# B&R Automation Studio project CControl_Gschneitner (part 16)

#### actionUpdateStatus.st
```iecst
ACTION actionUpdateStatus:

	//Sensoren *******************************************************************************************************************************************************************************
	gStatusAnlage.FrischluftTemperatur	:= aiFrischluftTemperatur;
	gStatusAnlage.FrischluftFeuchte		:= aiFrischluftFeuchte;
	gStatusAnlage.TrockenluftTemperatur	:= aiTrockenluftTemperatur;
	gStatusAnlage.TrockenluftFeuchte	:= aiTrockenluftFeuchte;
	gStatusAnlage.AbluftFeuchte			:= aiAbluftFeuchte;
	gStatusAnlage.AbluftTemperatur		:= aiAbluftTemperatur;
	gStatusAnlage.AustrittFeuchte		:= aiAustrittFeuchte;
	gStatusAnlage.AustrittTemperatur	:= aiAustrittTemperatur;
	gStatusAnlage.DachluftFeuchte		:= aiDachluftFeuchte;
	gStatusAnlage.DachluftTemperatur	:= aiDachluftTemperatur;
	gStatusAnlage.EintrittFeuchte		:= aiEintrittFeuchte;
	gStatusAnlage.EintrittTemperatur	:= aiEintrittTemperatur;
	gStatusAnlage.HochdruckModul1		:= aiHochdruckModul1;
	gStatusAnlage.HochdruckModul2		:= aiHochdruckModul2;
	gStatusAnlage.NiederdruckModul1		:= aiNiederdruckModul1;
	gStatusAnlage.NiederdruckModul2		:= aiNiederdruckModul2;
	gStatusAnlage.Luftgeschwindigkeit	:= aiLuftgeschwindigkeit;
	gStatusAnlage.Kanaldruck			:= aiDifferenzdruck;

	//Drehzahlvorgaben *********************************************************************************************************************************************************************
	gStatusAnlage.DrehzahlKompressorModul1	:= aoDrehzahlvorgKompressorModul1;
	gStatusAnlage.DrehzahlKompressorModul2	:= aoDrehzahlvorgKompressorModul2;
	gStatusAnlage.DrehzahlVentilator1		:= aoDrehzahlvorgVentilator1;
	gStatusAnlage.DrehzahlVentilator2		:= aoDrehzahlvorgVentilator2;

	//Luftmenge Aktuell **********************************************************************************************************************************************************************
	IF Betriebsparameter.Ausstattung.Entfeuchter THEN
		gStatusAnlage.LuftmengeAktuell	:= aiLuftgeschwindigkeit * Betriebsparameter.Entfeuchter.Registerflaeche[Betriebsparameter.Entfeuchter.IndexType] * 3600;
	ELSE
		gStatusAnlage.LuftmengeAktuell	:= aiLuftgeschwindigkeit * Betriebsparameter.Allgemein.AnsaugflaecheVent * 3600;
	END_IF

	//Status Frischluftbetrieb / Umluftbetrieb *****************************************************************************************************************************************************
	IF (hmiStatus.NameSteuerung <> 4) AND (hmiStatus.NameSteuerung <> 5) THEN
		gStatusAnlage.FrischluftbetriebAktiv	:= (fbEntfUmschaltung_0.FrischluftbetriebOut AND Betriebsparameter.Umschaltklappen.Automatik) OR
		Betriebsparameter.Umschaltklappen.Frischluft;
		gStatusAnlage.UmluftbetriebAktiv		:= (fbEntfUmschaltung_0.UmluftbetriebOut AND Betriebsparameter.Umschaltklappen.Automatik) OR
		Betriebsparameter.Umschaltklappen.Umluft;
	ELSE
		gStatusAnlage.FrischluftbetriebAktiv	:= (Betriebsparameter.Umschaltklappen.Automatik AND NOT gStatusAnlage.WetterIstSchlecht) OR
		Betriebsparameter.Umschaltklappen.Frischluft;
		gStatusAnlage.UmluftbetriebAktiv		:= (Betriebsparameter.Umschaltklappen.Automatik AND gStatusAnlage.WetterIstSchlecht) OR
		Betriebsparameter.Umschaltklappen.Umluft;
	END_IF

	//Status Warmluftanforderung (Kunde Gschneitner) ***************************************************************************************************************************
	//Warmluft = Umluftklappe des jeweiligen Ventilators angesteuert (dig. Ausgang logisch 1), Kaltluft = Klappe stromlos (logisch 0).
	//Es zaehlen nur laufende Ventilatoren: steht kein laufender Ventilator auf Warmluft, wird das Heizregister wie im Stillstand behandelt.
	gStatusAnlage.Warmluft1 := hmiButtons.changeWarmluftVent1;
	gStatusAnlage.Warmluft2 := hmiButtons.changeWarmluftVent2;
	gStatusAnlage.WarmluftAnforderung := (Aktoren.VentUndKlappen.FreigabeVentilator1Out AND gStatusAnlage.Warmluft1) OR
	(Aktoren.VentUndKlappen.FreigabeVentilator2Out AND gStatusAnlage.Warmluft2);

END_ACTION
```

#### actionStillstand.st
```iecst
ACTION actionStillstand:

	gStatusAnlage.Aktor[AKTOR_SCHRITTKETTE]	:= STATUS_STILLSTAND;

	//Notstromaggregat anfordern, wenn Notbetrieb Ventilatoren noch aktiv
	Aktoren.Notstromaggregat.NotstromaggregatAngefordert := (Boxen.NotbetriebVentilator1 OR Boxen.NotbetriebVentilator2) AND
	Betriebsparameter.Ausstattung.Notstromaggregat;

	//Ölsumpfheizungen Ein, wenn Entfeuchter in Ausstattung vorhanden
	Aktoren.OelsumpfheizungModul1.Freigabe			:= Betriebsparameter.Ausstattung.Entfeuchter;
	Aktoren.OelsumpfheizungModul2.Freigabe			:= Betriebsparameter.Ausstattung.Entfeuchter AND gModul2Vorhanden;

	//Luftentfeuchter AUS
	Aktoren.KompressorModul1.Freigabe			:= FALSE;
	Aktoren.KompressorModul1.Dauerbetrieb		:= FALSE;
	Aktoren.KompressorModul1.Automatik			:= FALSE;
	Aktoren.KompressorModul1.DrehzahlvorgabeFU	:= gCmdAnlage.Leistung.DrehzahlKompressorModul1;
	Aktoren.KompressorModul2.Freigabe			:= FALSE;
	Aktoren.KompressorModul2.Dauerbetrieb		:= FALSE;
	Aktoren.KompressorModul2.Automatik			:= FALSE;
	Aktoren.KompressorModul2.DrehzahlvorgabeFU	:= gCmdAnlage.Leistung.DrehzahlKompressorModul2;

	//Entfeuchter Fremdgerät AUS
	Aktoren.EntfeuchterFremd.Freigabe		:= FALSE;
	Aktoren.EntfeuchterFremd.Dauerbetrieb	:= FALSE;
	Aktoren.EntfeuchterFremd.Automatik		:= FALSE;

	//Ventilatoren 1 freigeben bei Notbetrieb (Trocknungsgeräte noch aktiv)
	IF (Aktoren.Notstromaggregat.NotstromBereitOut OR (NOT Betriebsparameter.Ausstattung.Notstromaggregat)) THEN
		Aktoren.VentUndKlappen.AnforderungVentilator1	:= Boxen.NotbetriebVentilator1;
		Aktoren.VentUndKlappen.DrehzahlVent1Betrieb		:= gCmdAnlage.Leistung.DrehzahlVentilator1;
	END_IF

	//Ventilatoren 2 freigeben bei Notbetrieb (Trocknungsgeräte noch aktiv)
	IF (Aktoren.Notstromaggregat.NotstromBereitOut OR (NOT Betriebsparameter.Ausstattung.Notstromaggregat)) THEN
		Aktoren.VentUndKlappen.AnforderungVentilator2	:= Boxen.NotbetriebVentilator2;
		Aktoren.VentUndKlappen.DrehzahlVent2Betrieb		:= gCmdAnlage.Leistung.DrehzahlVentilator2;
	END_IF

	//Warmluftofen AUS
	Aktoren.Warmluftofen.Freigabe			:= Betriebsparameter.Ausstattung.Warmluftofen;
	Aktoren.Warmluftofen.Automatikbetrieb	:= FALSE;
	Aktoren.Warmluftofen.Dauerbetrieb		:= FALSE;

	//Heizregister AUS
	Aktoren.Heizregister.Freigabe					:= Betriebsparameter.Ausstattung.Heizregister;
	Aktoren.Heizregister.Automatikbetrieb			:= FALSE;
	Aktoren.Heizregister.Dauerbetrieb				:= FALSE;
	Aktoren.Heizregister.DrehzahlHeizregisterSoll	:= gCmdAnlage.Leistung.DrehzahlHeizregister;

	//Abluftklappe Handbetrieb
	Aktoren.Abluftklappe.Freigabe			:= Betriebsparameter.Ausstattung.Abluftklappe;
	Aktoren.Abluftklappe.Automatik			:= FALSE;
	Aktoren.Abluftklappe.Oeffnen			:= Betriebsparameter.Abluftklappe.Oeffnen;
	Aktoren.Abluftklappe.Schliessen			:= Betriebsparameter.Abluftklappe.Schliessen;

	//Abluftventilator ein, wenn Ventilator noch in Betrieb
	Aktoren.Abluftventilator.Freigabe		:= Betriebsparameter.Ausstattung.Abluftventilator AND
	(Aktoren.VentUndKlappen.Ventilator1InBetrieb OR Aktoren.VentUndKlappen.Ventilator2InBetrieb);
	Aktoren.Abluftventilator.Automatik		:= Betriebsparameter.Abluftventilator.Automatik;
	Aktoren.Abluftventilator.Ein			:= Betriebsparameter.Abluftventilator.Ein;
	Aktoren.Abluftventilator.DrehzahlSoll	:= gCmdAnlage.Leistung.DrehzahlAbluftventilator;

	//Brandschutzklappe freigeben, wenn in Ausstattung vorhanden und WLO/SHO in Betrieb
	Aktoren.Brandschutzklappe.Oeffnen		:= Betriebsparameter.Ausstattung.Brandschutzklappe AND
	(Aktoren.Warmluftofen.WarmluftofenAktiv OR Aktoren.Scheitholzofen.ScheitholzofenAktiv);
	Aktoren.Brandschutzklappe.Schliessen	:= NOT Aktoren.Brandschutzklappe.Oeffnen;

	//Bypassklappe Handbetrieb
	Aktoren.VentUndKlappen.BypassklappeOeffnen		:= Betriebsparameter.Ausstattung.Bypassklappe AND
	(Betriebsparameter.Bypassklappe.Automatik OR Betriebsparameter.Bypassklappe.Oeffnen);
	Aktoren.VentUndKlappen.BypassklappeSchliessen	:= Betriebsparameter.Ausstattung.Bypassklappe AND Betriebsparameter.Bypassklappe.Schliessen;

	//Umschaltklappen Handbetrieb
	//Kunde Gschneitner: Warmluft-/Kaltluftumschaltung bleibt auch im Stillstand in der vom Bediener gewaehlten Stellung,
	//weil der digitale Ausgang der Klappe unveraendert dem HMI-Button folgt.
	IF Betriebsparameter.Ausstattung.Umschaltklappe1 OR Betriebsparameter.Ausstattung.Umschaltklappe2 THEN
		Aktoren.VentUndKlappen.Umschaltkl1Oeffnen		:= Betriebsparameter.Ausstattung.Umschaltklappe1 AND gStatusAnlage.Warmluft1;
		Aktoren.VentUndKlappen.Umschaltkl1Schliessen	:= Betriebsparameter.Ausstattung.Umschaltklappe1 AND NOT gStatusAnlage.Warmluft1;
		Aktoren.VentUndKlappen.Umschaltkl2Oeffnen		:= Betriebsparameter.Ausstattung.Umschaltklappe2 AND gStatusAnlage.Warmluft2;
		Aktoren.VentUndKlappen.Umschaltkl2Schliessen	:= Betriebsparameter.Ausstattung.Umschaltklappe2 AND NOT gStatusAnlage.Warmluft2;
	ELSE
		Aktoren.VentUndKlappen.Umschaltkl1Schliessen		:= FALSE;
		Aktoren.VentUndKlappen.Umschaltkl2Schliessen		:= FALSE;
		Aktoren.VentUndKlappen.Umschaltkl1Oeffnen			:= FALSE;
		Aktoren.VentUndKlappen.Umschaltkl2Oeffnen			:= FALSE;
	END_IF

	//Originallogik (Stellung je nach Betriebsart / Ausstattungsmenue) - fuer Kunde Gschneitner nicht in Verwendung:
	(*
	//Umschaltklappen Handbetrieb
	IF Betriebsparameter.Ausstattung.Umschaltklappe1 OR Betriebsparameter.Ausstattung.Umschaltklappe2 THEN
		//Stellung Umluftklappen je nach Einstellung im Ausstattungsmenü
		IF Betriebsparameter.Umschaltklappen.Automatik THEN
			Aktoren.VentUndKlappen.Umschaltkl1Schliessen	:= Betriebsparameter.Ausstattung.Umschaltklappe1 AND Betriebsparameter.Ausstattung.StellungUmluftklappe1Stillstand;
			Aktoren.VentUndKlappen.Umschaltkl2Schliessen	:= Betriebsparameter.Ausstattung.Umschaltklappe2 AND Betriebsparameter.Ausstattung.StellungUmluftklappe2Stillstand;
			Aktoren.VentUndKlappen.Umschaltkl1Oeffnen		:= Betriebsparameter.Ausstattung.Umschaltklappe1 AND NOT Betriebsparameter.Ausstattung.StellungUmluftklappe1Stillstand;
			Aktoren.VentUndKlappen.Umschaltkl2Oeffnen		:= Betriebsparameter.Ausstattung.Umschaltklappe2 AND NOT Betriebsparameter.Ausstattung.StellungUmluftklappe2Stillstand;
		ELSIF Betriebsparameter.Umschaltklappen.Frischluft THEN
			Aktoren.VentUndKlappen.Umschaltkl1Schliessen	:= Betriebsparameter.Ausstattung.Umschaltklappe1;
			Aktoren.VentUndKlappen.Umschaltkl2Schliessen	:= Betriebsparameter.Ausstattung.Umschaltklappe2;
			Aktoren.VentUndKlappen.Umschaltkl1Oeffnen		:= FALSE;
			Aktoren.VentUndKlappen.Umschaltkl2Oeffnen		:= FALSE;
		ELSIF Betriebsparameter.Umschaltklappen.Umluft THEN
			Aktoren.VentUndKlappen.Umschaltkl1Schliessen	:= FALSE;
			Aktoren.VentUndKlappen.Umschaltkl2Schliessen	:= FALSE;
			Aktoren.VentUndKlappen.Umschaltkl1Oeffnen		:= Betriebsparameter.Ausstattung.Umschaltklappe1;
			Aktoren.VentUndKlappen.Umschaltkl2Oeffnen		:= Betriebsparameter.Ausstattung.Umschaltklappe2;
		END_IF
	ELSE
		Aktoren.VentUndKlappen.Umschaltkl1Schliessen		:= FALSE;
		Aktoren.VentUndKlappen.Umschaltkl2Schliessen		:= FALSE;
		Aktoren.VentUndKlappen.Umschaltkl1Oeffnen			:= FALSE;
		Aktoren.VentUndKlappen.Umschaltkl2Oeffnen			:= FALSE;
	END_IF
	*)

END_ACTION
```

#### actionBetrieb.st
```iecst
ACTION actionBetrieb:

	gStatusAnlage.Aktor[AKTOR_SCHRITTKETTE]	:= STATUS_ANLAGE_IN_BETRIEB;

	//Notstromaggregat anfordern, wenn in Box in Betrieb und in Ausstattung vorhanden
	Aktoren.Notstromaggregat.NotstromaggregatAngefordert := (Boxen.Box1Out.BoxAktiv OR Boxen.Box2Out.BoxAktiv OR Boxen.Box3Out.BoxAktiv OR
	Boxen.Box4Out.BoxAktiv OR Boxen.Box5Out.BoxAktiv OR Boxen.Box6Out.BoxAktiv OR Boxen.NotbetriebBox1 OR Boxen.NotbetriebBox2 OR
	Boxen.NotbetriebBox3 OR Boxen.NotbetriebBox4 OR Boxen.NotbetriebBox5 OR Boxen.NotbetriebBox6 OR Boxen.NotbetriebVentilator1 OR Boxen.NotbetriebVentilator2)
	AND Betriebsparameter.Ausstattung.Notstromaggregat;

	//Ölsumpfheizungen Ein, wenn Kompressoren nicht in Betrieb (und Entfeuchter in Ausstattung vorhanden)
	Aktoren.OelsumpfheizungModul1.Freigabe			:= Betriebsparameter.Ausstattung.Entfeuchter AND NOT Aktoren.KompressorModul1.FreigabeKompressorOut;
	Aktoren.OelsumpfheizungModul2.Freigabe			:= Betriebsparameter.Ausstattung.Entfeuchter AND NOT Aktoren.KompressorModul2.FreigabeKompressorOut;

	//Luftentfeuchter freigeben, wenn von Boxen angefordert und Mindestlaufzeit Ölsumpfheizung abgelaufen und Notstromaggregat bereit und Ventilator bereit
	IF (gMindestlaufzOelsumpfOk OR ((hmiStatus.CurUserLevel > 2) AND (Nutzungsdaten.BstGes.Kompressor1Std < CONST_ZEIT_TESTPHASE))) AND
		(Aktoren.Notstromaggregat.NotstromBereitOut OR (NOT Betriebsparameter.Ausstattung.Notstromaggregat)) THEN

		Aktoren.KompressorModul1.Freigabe			:= Betriebsparameter.Ausstattung.Entfeuchter AND (Boxen.FreigabeLuftentfeuchter OR Boxen.FreigabeEntfeuchterInselbetrieb) AND
		((Boxen.EntfeuchterVonVent1Abhaengig AND Boxen.FreigabeVentilator1 (*Aktoren.VentUndKlappen.FreigabeVentilator1Out*) AND NOT Aktoren.VentUndKlappen.FehlerFuVentilator1) OR
		(Boxen.EntfeuchterVonVent2Abhaengig AND Boxen.FreigabeVentilator2 (*Aktoren.VentUndKlappen.FreigabeVentilator2Out*) AND NOT Aktoren.VentUndKlappen.FehlerFuVentilator2) OR
		(Boxen.FreigabeEntfeuchterInselbetrieb AND Aktoren.VentUndKlappen.Ventilator1InBetrieb)) AND NOT
		gCmdAnlage.FehlerModul1 AND (gStatusAnlage.UmluftbetriebAktiv OR (NOT Betriebsparameter.Ausstattung.EntfeuchterNurImUmluftbetrieb)) AND NOT
		Tarifabschaltung.TarifabschaltungLuftaufbEin;
		Aktoren.KompressorModul1.Dauerbetrieb		:= Betriebsparameter.Entfeuchter.Dauerbetrieb OR Boxen.FreigabeEntfeuchterInselbetrieb;
		Aktoren.KompressorModul1.Automatik			:= Betriebsparameter.Entfeuchter.Automatikbetrieb AND NOT Boxen.FreigabeEntfeuchterInselbetrieb;
		Aktoren.KompressorModul1.DrehzahlvorgabeFU	:= gCmdAnlage.Leistung.DrehzahlKompressorModul1;

		Aktoren.KompressorModul2.Freigabe			:= (Betriebsparameter.Ausstattung.Entfeuchter AND gModul2Vorhanden) AND (Boxen.FreigabeLuftentfeuchter OR Boxen.FreigabeEntfeuchterInselbetrieb) AND
		((Boxen.EntfeuchterVonVent1Abhaengig AND Boxen.FreigabeVentilator1 (*Aktoren.VentUndKlappen.FreigabeVentilator1Out*) AND NOT Aktoren.VentUndKlappen.FehlerFuVentilator1) OR
		(Boxen.EntfeuchterVonVent2Abhaengig AND Boxen.FreigabeVentilator2 (*Aktoren.VentUndKlappen.FreigabeVentilator2Out*) AND NOT Aktoren.VentUndKlappen.FehlerFuVentilator2) OR
		(Boxen.FreigabeEntfeuchterInselbetrieb AND Aktoren.VentUndKlappen.Ventilator1InBetrieb)) AND NOT
		gCmdAnlage.FehlerModul2 AND (gStatusAnlage.UmluftbetriebAktiv OR (NOT Betriebsparameter.Ausstattung.EntfeuchterNurImUmluftbetrieb)) AND NOT
		Tarifabschaltung.TarifabschaltungLuftaufbEin;;
		Aktoren.KompressorModul2.Dauerbetrieb		:= Betriebsparameter.Entfeuchter.Dauerbetrieb OR Boxen.FreigabeEntfeuchterInselbetrieb;
		Aktoren.KompressorModul2.Automatik			:= Betriebsparameter.Entfeuchter.Automatikbetrieb AND NOT Boxen.FreigabeEntfeuchterInselbetrieb;
		Aktoren.KompressorModul2.DrehzahlvorgabeFU	:= gCmdAnlage.Leistung.DrehzahlKompressorModul2;
	END_IF

	//Entfeuchter Fremdgerät freigeben, wenn Notstromaggregat bereit (oder kein Notstromaggregat vorhanden)
	IF (Aktoren.Notstromaggregat.NotstromBereitOut OR (NOT Betriebsparameter.Ausstattung.Notstromaggregat)) THEN
		Aktoren.EntfeuchterFremd.Freigabe			:= (Boxen.FreigabeLuftentfeuchter OR Boxen.FreigabeEntfeuchterInselbetrieb) AND
		((Boxen.EntfeuchterVonVent1Abhaengig AND Boxen.FreigabeVentilator1 AND NOT Aktoren.VentUndKlappen.FehlerFuVentilator1) OR
		(Boxen.EntfeuchterVonVent2Abhaengig AND Boxen.FreigabeVentilator2 AND NOT Aktoren.VentUndKlappen.FehlerFuVentilator2) OR
		(Boxen.FreigabeEntfeuchterInselbetrieb AND Aktoren.VentUndKlappen.Ventilator1InBetrieb)) AND NOT
		gCmdAnlage.FehlerModul1 AND (gStatusAnlage.UmluftbetriebAktiv OR (NOT Betriebsparameter.Ausstattung.EntfeuchterNurImUmluftbetrieb)) AND NOT
		Tarifabschaltung.TarifabschaltungLuftaufbEin;
		Aktoren.EntfeuchterFremd.Dauerbetrieb		:= Betriebsparameter.Entfeuchter.Dauerbetrieb OR Boxen.FreigabeEntfeuchterInselbetrieb;
		Aktoren.EntfeuchterFremd.Automatik			:= Betriebsparameter.Entfeuchter.Automatikbetrieb AND NOT Boxen.FreigabeEntfeuchterInselbetrieb;
	ELSE
		Aktoren.EntfeuchterFremd.Freigabe		:= FALSE;
		Aktoren.EntfeuchterFremd.Dauerbetrieb	:= FALSE;
		Aktoren.EntfeuchterFremd.Automatik		:= FALSE;
	END_IF

	//Ventilatoren 1 freigeben, wenn von Boxen angefordert und keine Tarifabschaltung (ausgenommen bei Notbetrieb wenn Trocknungsgeräte noch aktiv)
	IF (Aktoren.Notstromaggregat.NotstromBereitOut OR (NOT Betriebsparameter.Ausstattung.Notstromaggregat)) THEN
		Aktoren.VentUndKlappen.AnforderungVentilator1	:= (Boxen.FreigabeVentilator1 OR Boxen.NotbetriebVentilator1) AND NOT
		(Tarifabschaltung.TarifabschaltungEin AND NOT Boxen.NotbetriebVentilator1);
		Aktoren.VentUndKlappen.DrehzahlVent1Betrieb		:= gCmdAnlage.Leistung.DrehzahlVentilator1;
	ELSE
		Aktoren.VentUndKlappen.AnforderungVentilator1	:= FALSE;
	END_IF

	//Ventilatoren 2 freigeben, wenn von Boxen angefordert und keine Tarifabschaltung (ausgenommen bei Notbetrieb wenn Trocknungsgeräte noch aktiv)
	IF (Aktoren.Notstromaggregat.NotstromBereitOut OR (NOT Betriebsparameter.Ausstattung.Notstromaggregat)) THEN
		Aktoren.VentUndKlappen.AnforderungVentilator2	:= (Boxen.FreigabeVentilator2 OR Boxen.NotbetriebVentilator2) AND NOT
		(Tarifabschaltung.TarifabschaltungEin AND NOT Boxen.NotbetriebVentilator2);
		Aktoren.VentUndKlappen.DrehzahlVent2Betrieb		:= gCmdAnlage.Leistung.DrehzahlVentilator2;
	ELSE
		Aktoren.VentUndKlappen.AnforderungVentilator2	:= FALSE;
	END_IF

	//Warmluftofen freigeben, wenn von Boxen angefordert und Ventilator in Betrieb
	Aktoren.Warmluftofen.Freigabe			:= Betriebsparameter.Ausstattung.Warmluftofen AND Boxen.FreigabeWarmluftofen AND
	((Boxen.WarmluftofenVonVent1Abhaengig AND Aktoren.VentUndKlappen.FreigabeVentilator1Out AND NOT Aktoren.VentUndKlappen.FehlerFuVentilator1) OR
	(Boxen.WarmluftofenVonVent2Abhaengig AND Aktoren.VentUndKlappen.FreigabeVentilator2Out AND NOT Aktoren.VentUndKlappen.FehlerFuVentilator2)) AND NOT
	Tarifabschaltung.TarifabschaltungLuftaufbEin;
	Aktoren.Warmluftofen.Automatikbetrieb	:= Betriebsparameter.Warmluftofen.AutomatikbetriebEin;
	Aktoren.Warmluftofen.Dauerbetrieb		:= Betriebsparameter.Warmluftofen.DauerbetriebEin;

	//Heizregister freigeben, wenn von Boxen angefordert und zuständiger Ventilator aktiv
	Aktoren.Heizregister.Freigabe					:= Betriebsparameter.Ausstattung.Heizregister AND Boxen.FreigabeHeizregister  AND
	((Boxen.HeizregisterVonVent1Abhaengig AND Aktoren.VentUndKlappen.FreigabeVentilator1Out AND NOT Aktoren.VentUndKlappen.FehlerFuVentilator1) OR
	(Boxen.HeizregisterVonVent2Abhaengig AND Aktoren.VentUndKlappen.FreigabeVentilator2Out AND NOT Aktoren.VentUndKlappen.FehlerFuVentilator2)) AND NOT
	Tarifabschaltung.TarifabschaltungLuftaufbEin;
	Aktoren.Heizregister.Automatikbetrieb			:= Betriebsparameter.Heizregister.AutomatikbetriebEin;
	Aktoren.Heizregister.Dauerbetrieb				:= Betriebsparameter.Heizregister.DauerbetriebEin;
	Aktoren.Heizregister.DrehzahlHeizregisterSoll	:= gCmdAnlage.Leistung.DrehzahlHeizregister;

	//Kunde Gschneitner: Heizregister abschalten, wenn kein laufender Ventilator auf Warmluft steht.
	//Der Baustein wird dabei exakt wie im Stillstand versorgt -> FreigabeHeizregisterOut = FALSE und DrehzahlHeizregisterOut = 0.0.
	IF NOT gStatusAnlage.WarmluftAnforderung THEN
		Aktoren.Heizregister.Automatikbetrieb			:= FALSE;
		Aktoren.Heizregister.Dauerbetrieb				:= FALSE;
		Aktoren.Heizregister.DrehzahlHeizregisterSoll	:= 0.0;
	END_IF

	//Abluftklappe freigeben, wenn in Ausstattung vorhanden
	Aktoren.Abluftklappe.Freigabe			:= Betriebsparameter.Ausstattung.Abluftklappe;
	Aktoren.Abluftklappe.Automatik			:= Betriebsparameter.Abluftklappe.Automatik AND NOT
	(gStatusAnlage.FrischluftbetriebAktiv AND Betriebsparameter.Ausstattung.AbluftklImFrischlbetrImmerOffen);
	Aktoren.Abluftklappe.Oeffnen			:= Betriebsparameter.Abluftklappe.Oeffnen OR
	(gStatusAnlage.FrischluftbetriebAktiv AND Betriebsparameter.Ausstattung.AbluftklImFrischlbetrImmerOffen AND NOT Betriebsparameter.Abluftklappe.Schliessen);
	Aktoren.Abluftklappe.Schliessen			:= Betriebsparameter.Abluftklappe.Schliessen;

	//Abluftventilator freigeben, wenn in Ausstattung vorhanden
	Aktoren.Abluftventilator.Freigabe		:= Betriebsparameter.Ausstattung.Abluftventilator;
	Aktoren.Abluftventilator.Automatik		:= Betriebsparameter.Abluftventilator.Automatik AND (Boxen.Box1Out.BoxAktiv OR Boxen.Box2Out.BoxAktiv OR
	Boxen.Box3Out.BoxAktiv OR Boxen.Box4Out.BoxAktiv OR Boxen.Box5Out.BoxAktiv OR Boxen.Box6Out.BoxAktiv) AND NOT
	(gStatusAnlage.FrischluftbetriebAktiv AND Betriebsparameter.Ausstattung.AbluftklImFrischlbetrImmerOffen);
	Aktoren.Abluftventilator.Ein			:= Betriebsparameter.Abluftventilator.Ein OR
	(gStatusAnlage.FrischluftbetriebAktiv AND Betriebsparameter.Ausstattung.AbluftklImFrischlbetrImmerOffen AND (Boxen.Box1Out.BoxAktiv OR Boxen.Box2Out.BoxAktiv OR
	Boxen.Box3Out.BoxAktiv OR Boxen.Box4Out.BoxAktiv OR Boxen.Box5Out.BoxAktiv OR Boxen.Box6Out.BoxAktiv));
	Aktoren.Abluftventilator.DrehzahlSoll	:= gCmdAnlage.Leistung.DrehzahlAbluftventilator;

	//Brandschutzklappe freigeben, wenn in Ausstattung vorhanden und WLO/SHO in Betrieb
	Aktoren.Brandschutzklappe.Oeffnen		:= Betriebsparameter.Ausstattung.Brandschutzklappe AND
	(Aktoren.Warmluftofen.WarmluftofenAktiv OR Aktoren.Scheitholzofen.ScheitholzofenAktiv);
	Aktoren.Brandschutzklappe.Schliessen	:= NOT Aktoren.Brandschutzklappe.Oeffnen;

	//Bypassklappe freigeben, wenn in Ausstattung vorhanden
	IF Betriebsparameter.Bypassklappe.Automatik AND Betriebsparameter.Ausstattung.Bypassklappe AND NOT Betriebsparameter.Ausstattung.EntfeuchterFremd THEN
		IF NOT Aktoren.KompressorModul1.Freigabe AND NOT Aktoren.KompressorModul2.Freigabe THEN
			Aktoren.VentUndKlappen.BypassklappeOeffnen		:= TRUE;
			Aktoren.VentUndKlappen.BypassklappeSchliessen	:= FALSE;
		ELSE
			Aktoren.VentUndKlappen.BypassklappeOeffnen		:=  NOT Aktoren.KompressorModul1.loc_StatusFeuchteOk AND NOT Aktoren.KompressorModul2.loc_StatusFeuchteOk;
			Aktoren.VentUndKlappen.BypassklappeSchliessen	:= Aktoren.KompressorModul1.loc_StatusFeuchteOk OR Aktoren.KompressorModul2.loc_StatusFeuchteOk;
		END_IF
	//Ausstattung mit Entfeuchter Fremdgerät
	ELSIF Betriebsparameter.Bypassklappe.Automatik AND Betriebsparameter.Ausstattung.Bypassklappe THEN
		IF NOT Aktoren.EntfeuchterFremd.Freigabe THEN
			Aktoren.VentUndKlappen.BypassklappeOeffnen		:= TRUE;
			Aktoren.VentUndKlappen.BypassklappeSchliessen	:= FALSE;
		ELSE
			Aktoren.VentUndKlappen.BypassklappeOeffnen		:=  NOT Aktoren.EntfeuchterFremd.WitterungIstSchlecht;
			Aktoren.VentUndKlappen.BypassklappeSchliessen	:= Aktoren.EntfeuchterFremd.WitterungIstSchlecht;
		END_IF
	ELSE
		Aktoren.VentUndKlappen.BypassklappeOeffnen		:= Betriebsparameter.Ausstattung.Bypassklappe AND Betriebsparameter.Bypassklappe.Oeffnen;
		Aktoren.VentUndKlappen.BypassklappeSchliessen	:= Betriebsparameter.Ausstattung.Bypassklappe AND Betriebsparameter.Bypassklappe.Schliessen;
	END_IF
	(*
	Aktoren.VentUndKlappen.BypassklappeOeffnen		:= Betriebsparameter.Ausstattung.Bypassklappe AND (Betriebsparameter.Bypassklappe.Oeffnen OR
	(Betriebsparameter.Bypassklappe.Automatik AND NOT Aktoren.KompressorModul1.loc_StatusFeuchteOk AND NOT Aktoren.KompressorModul2.loc_StatusFeuchteOk));
	Aktoren.VentUndKlappen.BypassklappeSchliessen	:= Betriebsparameter.Ausstattung.Bypassklappe AND (Betriebsparameter.Bypassklappe.Schliessen OR
	(Betriebsparameter.Bypassklappe.Automatik AND (Aktoren.KompressorModul1.loc_StatusFeuchteOk OR Aktoren.KompressorModul2.loc_StatusFeuchteOk)));
	*)

	//Umschaltklappen je nach Betriebsart umschalten
	//Kunde Gschneitner: die Umschaltklappen werden als Warmluft-/Kaltluftumschaltung verwendet und direkt vom Bediener geschaltet.
	//Die Betriebsart ist fest auf Frischluft gestellt, deshalb entfaellt die witterungsgefuehrte Umschaltung.
	//Die Klappenbausteine werden hier mit der tatsaechlichen Stellung versorgt, damit Laufzeit-/Endlagenueberwachung und
	//die Statusanzeigen in der Visu mit dem realen Ausgang zusammenpassen.
	IF Betriebsparameter.Ausstattung.Umschaltklappe1 OR Betriebsparameter.Ausstattung.Umschaltklappe2 THEN
		Aktoren.VentUndKlappen.Umschaltkl1Oeffnen		:= Betriebsparameter.Ausstattung.Umschaltklappe1 AND gStatusAnlage.Warmluft1;
		Aktoren.VentUndKlappen.Umschaltkl1Schliessen	:= Betriebsparameter.Ausstattung.Umschaltklappe1 AND NOT gStatusAnlage.Warmluft1;
		Aktoren.VentUndKlappen.Umschaltkl2Oeffnen		:= Betriebsparameter.Ausstattung.Umschaltklappe2 AND gStatusAnlage.Warmluft2;
		Aktoren.VentUndKlappen.Umschaltkl2Schliessen	:= Betriebsparameter.Ausstattung.Umschaltklappe2 AND NOT gStatusAnlage.Warmluft2;
	ELSE
		Aktoren.VentUndKlappen.Umschaltkl1Schliessen		:= FALSE;
		Aktoren.VentUndKlappen.Umschaltkl2Schliessen		:= FALSE;
		Aktoren.VentUndKlappen.Umschaltkl1Oeffnen			:= FALSE;
		Aktoren.VentUndKlappen.Umschaltkl2Oeffnen			:= FALSE;
	END_IF

	//Originallogik (Betriebsart Automatik/Frischluft/Umluft) - fuer Kunde Gschneitner nicht in Verwendung:
	(*
	//Umschaltklappen je nach Betriebsart umschalten
	IF Betriebsparameter.Ausstattung.Umschaltklappe1 OR Betriebsparameter.Ausstattung.Umschaltklappe2 THEN
		//Konfiguration HB3000 und HB4000 -> Umschaltklappen nach Witterung umschalten (Kein eigener Schaltpunkt)
		IF (hmiStatus.NameSteuerung = 4) OR (hmiStatus.NameSteuerung = 5) THEN
			IF Betriebsparameter.Umschaltklappen.Frischluft OR (Betriebsparameter.Umschaltklappen.Automatik AND NOT gStatusAnlage.WetterIstSchlecht) THEN
				Aktoren.VentUndKlappen.Umschaltkl1Schliessen	:= Betriebsparameter.Ausstattung.Umschaltklappe1;
				Aktoren.VentUndKlappen.Umschaltkl2Schliessen	:= Betriebsparameter.Ausstattung.Umschaltklappe2;
				Aktoren.VentUndKlappen.Umschaltkl1Oeffnen		:= FALSE;
				Aktoren.VentUndKlappen.Umschaltkl2Oeffnen		:= FALSE;
			ELSIF Betriebsparameter.Umschaltklappen.Umluft OR (Betriebsparameter.Umschaltklappen.Automatik AND gStatusAnlage.WetterIstSchlecht) THEN
				Aktoren.VentUndKlappen.Umschaltkl1Schliessen	:= FALSE;
				Aktoren.VentUndKlappen.Umschaltkl2Schliessen	:= FALSE;
				Aktoren.VentUndKlappen.Umschaltkl1Oeffnen		:= Betriebsparameter.Ausstattung.Umschaltklappe1;
				Aktoren.VentUndKlappen.Umschaltkl2Oeffnen		:= Betriebsparameter.Ausstattung.Umschaltklappe2;
			END_IF
		ELSIF Betriebsparameter.Umschaltklappen.Frischluft OR (Betriebsparameter.Umschaltklappen.Automatik AND gStatusAnlage.FrischluftbetriebAktiv) THEN
			Aktoren.VentUndKlappen.Umschaltkl1Schliessen	:= Betriebsparameter.Ausstattung.Umschaltklappe1;
			Aktoren.VentUndKlappen.Umschaltkl2Schliessen	:= Betriebsparameter.Ausstattung.Umschaltklappe2;
			Aktoren.VentUndKlappen.Umschaltkl1Oeffnen		:= FALSE;
			Aktoren.VentUndKlappen.Umschaltkl2Oeffnen		:= FALSE;
		ELSIF Betriebsparameter.Umschaltklappen.Umluft OR (Betriebsparameter.Umschaltklappen.Automatik AND gStatusAnlage.UmluftbetriebAktiv) THEN
			Aktoren.VentUndKlappen.Umschaltkl1Schliessen	:= FALSE;
			Aktoren.VentUndKlappen.Umschaltkl2Schliessen	:= FALSE;
			Aktoren.VentUndKlappen.Umschaltkl1Oeffnen		:= Betriebsparameter.Ausstattung.Umschaltklappe1;
			Aktoren.VentUndKlappen.Umschaltkl2Oeffnen		:= Betriebsparameter.Ausstattung.Umschaltklappe2;
		END_IF
	ELSE
		Aktoren.VentUndKlappen.Umschaltkl1Schliessen		:= FALSE;
		Aktoren.VentUndKlappen.Umschaltkl2Schliessen		:= FALSE;
		Aktoren.VentUndKlappen.Umschaltkl1Oeffnen			:= FALSE;
		Aktoren.VentUndKlappen.Umschaltkl2Oeffnen			:= FALSE;
	END_IF
	*)

END_ACTION
```

### Package Logical/Steuerung - Generierung der Start- und Stoppsignale

### Program Logical/Steuerung/StartStopp (IEC) - Auswertung der Start- und Stoppsignale

#### StartStopp.st - Zyklischer Code
```iecst
PROGRAM _CYCLIC

	//Ticks erzeugen
	//==============
	fbLascoZdxx_0(IN	:= Echtzeit.Milli / 100);
	hmilliTick			:= fbLascoZdxx_0.Q;

	fbLascoPuge_0(StartMitPuls := TRUE, Tick := hmilliTick, ZeitPuls := 8, ZeitPause := 8,);
	hmiBlink			:= fbLascoPuge_0.PulsQ;

	//Automatik oder Testmodus
	//************************

	gCmdAnlage.Auto   		:= NOT hmiButtons.TestbetriebEin;
	gCmdAnlage.Test   		:= hmiButtons.TestbetriebEin;

	//Externe Start/Stopp- Signale
(*	gCmdAnlage.StartExtern		:= diAnfEntfeuchterExtern;
	gCmdAnlage.StoppExtern		:= NOT diAnfEntfeuchterExtern;*)

	//Start- und Stoppsignale auswerten
	//=================================

	//Startsignal geben, wenn eine der Boxen angefordert wird
	gCmdAnlage.Start	:= gCmdAnlage.Auto AND (Boxen.Box1Out.BoxBereit OR Boxen.Box2Out.BoxBereit OR Boxen.Box3Out.BoxBereit OR Boxen.Box4Out.BoxBereit OR
	Boxen.Box5Out.BoxBereit OR Boxen.Box6Out.BoxBereit OR Boxen.EntfeuchterInselbetrAktivOut);

	//Stopsignal geben, wenn keine Box angefordert ist
	gCmdAnlage.Stop		:= gCmdAnlage.Auto AND NOT Boxen.Box1Out.BoxBereit AND NOT Boxen.Box2Out.BoxBereit AND NOT Boxen.Box3Out.BoxBereit AND NOT Boxen.Box4Out.BoxBereit AND NOT
	Boxen.Box5Out.BoxBereit AND NOT Boxen.Box6Out.BoxBereit AND NOT Boxen.EntfeuchterInselbetrAktivOut;

	//Signal Fehler-Stopp erzeugen (kein Start möglich bzw. Abbruch Trocknung)
	//Fehlerstopp entfernt (Trocknung lässt sich dennoch starten, je nach Fehler werden die einzelnen Aktoren nicht freigegeben
	gCmdAnlage.FehlerStopp	:= FALSE;
(*	gCmdAnlage.FehlerStopp	:= (gCmdAnlage.Auto AND (alarmFehler[FEHLER_24VDC] OR alarmFehler[FEHLER_ENDLAGEN_BOXENKLAPPE_1] OR
	alarmFehler[FEHLER_ENDLAGEN_BOXENKLAPPE_2] OR alarmFehler[FEHLER_ENDLAGEN_BOXENKLAPPE_3] OR alarmFehler[FEHLER_ENDLAGEN_BOXENKLAPPE_4] OR
	alarmFehler[FEHLER_ENDLAGEN_BOXENKLAPPE_5] OR alarmFehler[FEHLER_ENDLAGEN_BOXENKLAPPE_6] OR alarmFehler[FEHLER_ENDLAGEN_BYPASSKLAPPE] OR
	alarmFehler[FEHLER_ENDLAGEN_UMSCHALTKLAPPE1] OR alarmFehler[FEHLER_ENDLAGEN_UMSCHALTKLAPPE2] OR alarmFehler[FEHLER_IO_TEST_NICHT_FERTIG] OR
	alarmFehler[FEHLER_KOMMUNIKATION_DISPLAY_IO] OR alarmFehler[FEHLER_BETRIEBSMLDG_NOTSTROM] OR alarmFehler[FEHLER_BETRIEBSMLDG_VENTILATOR1] OR
	alarmFehler[FEHLER_BETRIEBSMLDG_VENTILATOR2]));

	//Bei Doppelmodulen Anlage nur stoppen, wenn bei beiden Modulen ein Fehler anliegt
	IF gModul2Vorhanden THEN
		gCmdAnlage.FehlerStopp := (gCmdAnlage.Auto AND (alarmFehler[FEHLER_24VDC] OR alarmFehler[FEHLER_ENDLAGEN_BOXENKLAPPE_1] OR alarmFehler[FEHLER_ENDLAGEN_BOXENKLAPPE_2] OR
		alarmFehler[FEHLER_ENDLAGEN_BOXENKLAPPE_3] OR alarmFehler[FEHLER_ENDLAGEN_BOXENKLAPPE_4] OR alarmFehler[FEHLER_ENDLAGEN_BOXENKLAPPE_5] OR
		alarmFehler[FEHLER_ENDLAGEN_BOXENKLAPPE_6] OR alarmFehler[FEHLER_ENDLAGEN_BYPASSKLAPPE] OR alarmFehler[FEHLER_ENDLAGEN_UMSCHALTKLAPPE1] OR
		alarmFehler[FEHLER_ENDLAGEN_UMSCHALTKLAPPE2] OR alarmFehler[FEHLER_IO_TEST_NICHT_FERTIG] OR alarmFehler[FEHLER_KOMMUNIKATION_DISPLAY_IO] OR
		alarmFehler[FEHLER_EINTRITT_TEMP_ZU_HOCH] OR alarmFehler[FEHLER_EINTRITT_TEMP_ZU_NIEDRIG] OR (gCmdAnlage.FehlerModul1 AND gCmdAnlage.FehlerModul2)));
	ELSE
		gCmdAnlage.FehlerStopp := (gCmdAnlage.Auto AND (alarmFehler[FEHLER_24VDC] OR alarmFehler[FEHLER_ENDLAGEN_BOXENKLAPPE_1] OR alarmFehler[FEHLER_ENDLAGEN_BOXENKLAPPE_2] OR
		alarmFehler[FEHLER_ENDLAGEN_BOXENKLAPPE_3] OR alarmFehler[FEHLER_ENDLAGEN_BOXENKLAPPE_4] OR alarmFehler[FEHLER_ENDLAGEN_BOXENKLAPPE_5] OR
		alarmFehler[FEHLER_ENDLAGEN_BOXENKLAPPE_6] OR alarmFehler[FEHLER_ENDLAGEN_BYPASSKLAPPE] OR alarmFehler[FEHLER_ENDLAGEN_UMSCHALTKLAPPE1] OR
		alarmFehler[FEHLER_ENDLAGEN_UMSCHALTKLAPPE2] OR alarmFehler[FEHLER_IO_TEST_NICHT_FERTIG] OR alarmFehler[FEHLER_KOMMUNIKATION_DISPLAY_IO] OR
		alarmFehler[FEHLER_EINTRITT_TEMP_ZU_HOCH] OR alarmFehler[FEHLER_EINTRITT_TEMP_ZU_NIEDRIG] OR gCmdAnlage.FehlerModul1));
	END_IF
	*)
	//Fehler Modul 1
	gCmdAnlage.FehlerModul1	:= (gCmdAnlage.Auto AND (alarmFehler[FEHLER_BETRIEBSMLDG_KOMPR_MOD1] OR alarmFehler[FEHLER_FU_KOMPRESSOR_MODUL1] OR alarmFehler[FEHLER_HOCHDRUCK_MODUL1] OR
	alarmFehler[FEHLER_KOPFTEMP_KOMPR_MOD1] OR alarmFehler[FEHLER_NIEDERDRUCK_MODUL1] OR alarmFehler[FEHLER_OELDRUCK_KOMPR_MOD1] OR alarmFehler[FEHLER_SENSOR_HOCHDRUCK_MOD1] OR
	alarmFehler[FEHLER_SENSOR_NIEDERDRUCK_MOD1] OR alarmFehler[FEHLER_VOLLSCHUTZ_KOMPR_MOD1] OR alarmFehler[FEHLER_LZ_PUMPDOWN_MOD1] OR alarmFehler[FEHLER_DREHFELD] OR
	alarmFehler[FEHLER_ENTF_FREMD_BETRMLDG] OR alarmFehler[FEHLER_ENTF_FREMD_STOERMELDUNG])); //Ab V2.0.0: Fehler Entfeuchter Fremd hinzugefügt

	//Fehler Modul 2
	gCmdAnlage.FehlerModul2	:= (gCmdAnlage.Auto AND gModul2Vorhanden AND (alarmFehler[FEHLER_BETRIEBSMLDG_KOMPR_MOD2] OR alarmFehler[FEHLER_FU_KOMPRESSOR_MODUL2] OR alarmFehler[FEHLER_HOCHDRUCK_MODUL2] OR
	alarmFehler[FEHLER_KOPFTEMP_KOMPR_MOD2] OR alarmFehler[FEHLER_NIEDERDRUCK_MODUL2] OR alarmFehler[FEHLER_OELDRUCK_KOMPR_MOD2] OR alarmFehler[FEHLER_SENSOR_HOCHDRUCK_MOD2] OR
	alarmFehler[FEHLER_SENSOR_NIEDERDRUCK_MOD2] OR alarmFehler[FEHLER_VOLLSCHUTZ_KOMPR_MOD2] OR alarmFehler[FEHLER_LZ_PUMPDOWN_MOD2] OR alarmFehler[FEHLER_DREHFELD]));

	//Betriebsmeldung und Störmeldung
	gStatusAnlage.Betrieb	:= gAktModus = BETRIEB;

	IF gStatusAnlage.Betrieb AND (doVentilator1Ein OR doVentilator2Ein) THEN
		doTrocknungInBetrieb := TRUE;
	ELSIF gStatusAnlage.Betrieb AND (doKompressorEinModul1 OR doKompressorEinModul2) AND NOT Betriebsparameter.Ausstattung.Ventilator1 THEN
		doTrocknungInBetrieb := TRUE;
	ELSIF gStatusAnlage.Betrieb THEN
		doTrocknungInBetrieb := hmiBlink;
	ELSE
		doTrocknungInBetrieb := FALSE;
	END_IF

	doTrocknungStoerung		:= gStatusAnlage.Fehler.SummeFehler;

END_PROGRAM
```

#### StartStopp.var - Lokale Variablen
```iecst
VAR
	fbLascoZdxx_0 : {REDUND_UNREPLICABLE} fbLascoZdxx;
	hmilliTick : {REDUND_UNREPLICABLE} BOOL;
	fbLascoPuge_0 : {REDUND_UNREPLICABLE} fbLascoPuge;
	hmiBlink : {REDUND_UNREPLICABLE} BOOL;
END_VAR
```

### Package Logical/Regelung - Luftmengen- und Druckregler

### Program Logical/Regelung/Leistung (IEC) - Leistungsvorgabe an Ventilatoren

#### Leistung.st - Zyklischer Code
```iecst
PROGRAM _INIT

	//Luftmengenregler für Ventilator 1 initialisieren
	fbPidLuftmengeVent1.Mode	:= FBREG_MODUS_AUS;
	fbPidLuftmengeVent1();

	//Luftmengenregler für Ventilator 2 initialisieren
	fbPidLuftmengeVent2.Mode	:= FBREG_MODUS_AUS;
	fbPidLuftmengeVent2();

	//Regler Entfeuchter Kompressor 1 -Drehzahl initialisieren
	fbPidKompressor1.Mode	:= FBREG_MODUS_AUS;
	fbPidKompressor1();

	//Regler Entfeuchter Kompressor 2 -Drehzahl initialisieren
	fbPidKompressor2.Mode	:= FBREG_MODUS_AUS;
	fbPidKompressor2();

	//Regler Heizregister-Pumpe initialisieren
	fbPidHeizregister.Mode	:= FBREG_MODUS_AUS;
	fbPidHeizregister();

	//Abluftregler initialisieren
	fbPidAbluftregler.Mode		:= FBREG_MODUS_AUS;
	fbPidAbluftregler();

END_PROGRAM

PROGRAM _CYCLIC

	//Zeitticks erzeugen
	fbLascoZdxx_0(IN 	:= Echtzeit.Minute);
	minTick				:= fbLascoZdxx_0.Q;
	fbLascoZdxx_1(IN	:= Echtzeit.Sekunde);
	sekTick				:= fbLascoZdxx_1.Q;

	//Erforderliche Soll-Luftmengen für Ventilator 1 & 2 ermitteln
	//************************************************************

	fbBoxenLuftmengen_0.EntfeuchterInBetrieb			:= Aktoren.KompressorModul1.FreigabeKompressorOut OR Aktoren.KompressorModul2.FreigabeKompressorOut OR
	diEntfeuchterFremdInBetrieb;
	//Kunde Gschneitner: wird weiter unten je Parametersatz (Kalt-/Warmluft) ueberschrieben
	fbBoxenLuftmengen_0.FrischluftbetriebAktiv			:= gStatusAnlage.FrischluftbetriebAktiv;
	fbBoxenLuftmengen_0.UmluftbetriebAktiv				:= gStatusAnlage.UmluftbetriebAktiv;
	fbBoxenLuftmengen_0.LuftgeschwEntfeuchterMin		:= Betriebsparameter.Entfeuchter.LuftgeschwEntfeuchterMin;
	fbBoxenLuftmengen_0.LuftgeschwEntfeuchterMax		:= Betriebsparameter.Entfeuchter.LuftgeschwEntfeuchterMax;
	fbBoxenLuftmengen_0.LuftmengeSollProM2FrischlVent1	:= Betriebsparameter.Ventilator1.LuftmengeSollFrischluft;
	fbBoxenLuftmengen_0.LuftmengeSollProM2UmluftVent1	:= Betriebsparameter.Ventilator1.LuftmengeSollUmluft;
	fbBoxenLuftmengen_0.LuftmengeSollProM2FrischlVent2	:= Betriebsparameter.Ventilator2.LuftmengeSollFrischluft;
	fbBoxenLuftmengen_0.LuftmengeSollProM2UmluftVent2	:= Betriebsparameter.Ventilator2.LuftmengeSollUmluft;
	IF Betriebsparameter.Ausstattung.EntfeuchterFremd THEN
		fbBoxenLuftmengen_0.RegisterflaecheEntfeuchter		:= Betriebsparameter.Allgemein.AnsaugflaecheVent;
	ELSE
		fbBoxenLuftmengen_0.RegisterflaecheEntfeuchter		:= Betriebsparameter.Entfeuchter.Registerflaeche[Betriebsparameter.Entfeuchter.IndexType];
	END_IF

	fbBoxenLuftmengen_0.Box1.BoxIstAktiv		:= Boxen.Box1Out.BoxAktiv;
	fbBoxenLuftmengen_0.Box1.GrundflaecheBox	:= Betriebsparameter.Boxen[1].Grundflaeche;
	fbBoxenLuftmengen_0.Box1.Ventilator1		:= Betriebsparameter.Boxen[1].Ventilator1;
	fbBoxenLuftmengen_0.Box1.Ventilator2		:= Betriebsparameter.Boxen[1].Ventilator2;

	fbBoxenLuftmengen_0.Box2.BoxIstAktiv		:= Boxen.Box2Out.BoxAktiv;
	fbBoxenLuftmengen_0.Box2.GrundflaecheBox	:= Betriebsparameter.Boxen[2].Grundflaeche;
	fbBoxenLuftmengen_0.Box2.Ventilator1		:= Betriebsparameter.Boxen[2].Ventilator1;
	fbBoxenLuftmengen_0.Box2.Ventilator2		:= Betriebsparameter.Boxen[2].Ventilator2;

	fbBoxenLuftmengen_0.Box3.BoxIstAktiv		:= Boxen.Box3Out.BoxAktiv;
	fbBoxenLuftmengen_0.Box3.GrundflaecheBox	:= Betriebsparameter.Boxen[3].Grundflaeche;
	fbBoxenLuftmengen_0.Box3.Ventilator1		:= Betriebsparameter.Boxen[3].Ventilator1;
	fbBoxenLuftmengen_0.Box3.Ventilator2		:= Betriebsparameter.Boxen[3].Ventilator2;

	fbBoxenLuftmengen_0.Box4.BoxIstAktiv		:= Boxen.Box4Out.BoxAktiv;
	fbBoxenLuftmengen_0.Box4.GrundflaecheBox	:= Betriebsparameter.Boxen[4].Grundflaeche;
	fbBoxenLuftmengen_0.Box4.Ventilator1		:= Betriebsparameter.Boxen[4].Ventilator1;
	fbBoxenLuftmengen_0.Box4.Ventilator2		:= Betriebsparameter.Boxen[4].Ventilator2;

	fbBoxenLuftmengen_0.Box5.BoxIstAktiv		:= Boxen.Box5Out.BoxAktiv;
	fbBoxenLuftmengen_0.Box5.GrundflaecheBox	:= Betriebsparameter.Boxen[5].Grundflaeche;
	fbBoxenLuftmengen_0.Box5.Ventilator1		:= Betriebsparameter.Boxen[5].Ventilator1;
	fbBoxenLuftmengen_0.Box5.Ventilator2		:= Betriebsparameter.Boxen[5].Ventilator2;

	fbBoxenLuftmengen_0.Box6.BoxIstAktiv		:= Boxen.Box6Out.BoxAktiv;
	fbBoxenLuftmengen_0.Box6.GrundflaecheBox	:= Betriebsparameter.Boxen[6].Grundflaeche;
	fbBoxenLuftmengen_0.Box6.Ventilator1		:= Betriebsparameter.Boxen[6].Ventilator1;
	fbBoxenLuftmengen_0.Box6.Ventilator2		:= Betriebsparameter.Boxen[6].Ventilator2;

	//Kunde Gschneitner: Kaltluft entspricht dem frueheren Frischluftbetrieb, Warmluft dem Umluftbetrieb.
	//Die beiden Ventilatoren koennen unterschiedlich stehen, der Baustein kennt aber nur eine gemeinsame
	//Betriebsart. Er wird deshalb zweimal aufgerufen (er ist rein kombinatorisch, hat also keinen Zustand)
	//und beide Ergebnisse werden zwischengespeichert.
	fbBoxenLuftmengen_0.FrischluftbetriebAktiv			:= TRUE;
	fbBoxenLuftmengen_0.UmluftbetriebAktiv				:= FALSE;
	fbBoxenLuftmengen_0();
	loc_LuftmengeSollKaltVent1							:= fbBoxenLuftmengen_0.LuftmengeSollVent1Out;
	loc_LuftmengeSollKaltVent2							:= fbBoxenLuftmengen_0.LuftmengeSollVent2Out;

	fbBoxenLuftmengen_0.FrischluftbetriebAktiv			:= FALSE;
	fbBoxenLuftmengen_0.UmluftbetriebAktiv				:= TRUE;
	fbBoxenLuftmengen_0();
	loc_LuftmengeSollWarmVent1							:= fbBoxenLuftmengen_0.LuftmengeSollVent1Out;
	loc_LuftmengeSollWarmVent2							:= fbBoxenLuftmengen_0.LuftmengeSollVent2Out;

	//Erforderliche Luftmengen Ventilator 1 & 2 in Luftgeschwindigkeit umrechnen
	//**************************************************************************

	//Auswahl, ob Registerfläche oder Ansaugfläche zur Berechnung verwendet wird (Registerfläche nur wenn Entfeuchter vorhanden)
	IF Betriebsparameter.Ausstattung.Entfeuchter THEN
		loc_Ansaugflaeche	:= Betriebsparameter.Entfeuchter.Registerflaeche[Betriebsparameter.Entfeuchter.IndexType];
	ELSE
		loc_Ansaugflaeche	:= Betriebsparameter.Allgemein.AnsaugflaecheVent;
	END_IF

	//Kunde Gschneitner: Sollwert je nach Stellung der Warmluft-/Kaltluftumschaltung des jeweiligen Ventilators.
	//Warmluft verwendet die Umluftlogik (LuftmengeSollUmluft), Kaltluft die Frischluftlogik (LuftmengeSollFrischluft).
	//In der Ausstattung ist die Luftmengenregelung nur fuer Umluft (= Warmluft) freigegeben, im Kaltluftbetrieb
	//laeuft der Ventilator mit der Fixdrehzahl des Frischluftbetriebs.

	//Ventilator 1
	IF gStatusAnlage.Warmluft1 AND Betriebsparameter.Ventilator1.LuftmengenregUmluftEin THEN
		IF loc_Ansaugflaeche <> 0 THEN
			loc_LuftgeschwSollVent1	:= loc_LuftmengeSollWarmVent1 / loc_Ansaugflaeche / 3600;
		END_IF
	ELSIF (NOT gStatusAnlage.Warmluft1) AND Betriebsparameter.Ventilator1.LuftmengenregFrischluftEin THEN
		IF loc_Ansaugflaeche <> 0 THEN
			loc_LuftgeschwSollVent1	:= loc_LuftmengeSollKaltVent1 / loc_Ansaugflaeche / 3600;
		END_IF
	END_IF

	//Ventilator 2
	IF gStatusAnlage.Warmluft2 AND Betriebsparameter.Ventilator2.LuftmengenregUmluftEin THEN
		IF loc_Ansaugflaeche <> 0 THEN
			loc_LuftgeschwSollVent2	:= loc_LuftmengeSollWarmVent2 / loc_Ansaugflaeche / 3600;
		END_IF
	ELSIF (NOT gStatusAnlage.Warmluft2) AND Betriebsparameter.Ventilator2.LuftmengenregFrischluftEin THEN
		IF loc_Ansaugflaeche <> 0 THEN
			loc_LuftgeschwSollVent2	:= loc_LuftmengeSollKaltVent2 / loc_Ansaugflaeche / 3600;
		END_IF
	END_IF

	//Originallogik (Frischluft-/Umluftbetrieb) - fuer Kunde Gschneitner nicht in Verwendung:
	(*
	//Ventilator 1 - Frischluftbetrieb aktiv
	IF gStatusAnlage.FrischluftbetriebAktiv AND Betriebsparameter.Ventilator1.LuftmengenregFrischluftEin THEN
		IF loc_Ansaugflaeche <> 0 THEN
			loc_LuftgeschwSollVent1	:= fbBoxenLuftmengen_0.LuftmengeSollVent1Out / loc_Ansaugflaeche / 3600;
		END_IF
		//Ventilator 2 - Umluftbetrieb aktiv
	ELSIF gStatusAnlage.UmluftbetriebAktiv AND Betriebsparameter.Ventilator1.LuftmengenregUmluftEin THEN
		IF loc_Ansaugflaeche <> 0 THEN
			loc_LuftgeschwSollVent1	:= fbBoxenLuftmengen_0.LuftmengeSollVent1Out / loc_Ansaugflaeche / 3600;
		END_IF
	END_IF

	//Ventilator 2 - Frischluftbetrieb aktiv
	IF gStatusAnlage.FrischluftbetriebAktiv AND Betriebsparameter.Ventilator2.LuftmengenregFrischluftEin THEN
		IF loc_Ansaugflaeche <> 0 THEN
			loc_LuftgeschwSollVent2	:= fbBoxenLuftmengen_0.LuftmengeSollVent2Out / loc_Ansaugflaeche / 3600;
		END_IF
		//Ventilator 2 - Umluftbetrieb aktiv
	ELSIF gStatusAnlage.UmluftbetriebAktiv AND Betriebsparameter.Ventilator2.LuftmengenregUmluftEin THEN
		IF loc_Ansaugflaeche <> 0 THEN
			loc_LuftgeschwSollVent2	:= fbBoxenLuftmengen_0.LuftmengeSollVent2Out / loc_Ansaugflaeche / 3600;
		END_IF
	END_IF
	*)

	//====================================================================================================================================================================================
	//Luftmengenregler Ventilator 1 Eingänge
	//====================================================================================================================================================================================

	PidLuftmengeVent1.Sollgroesse				:= loc_LuftgeschwSollVent1;
	fbPidLuftmengeVent1.Freigabe				:= PidLuftmengeVent1.Enable;
	fbPidLuftmengeVent1.Sollwert				:= PidLuftmengeVent1.Sollgroesse;
	fbPidLuftmengeVent1.Istwert					:= gStatusAnlage.Luftgeschwindigkeit;
	fbPidLuftmengeVent1.AbschwaechungSollwert	:= 1.0;
	fbPidLuftmengeVent1.Aufschaltgroesse		:= 0.0;
	fbPidLuftmengeVent1.Fehlerverzoegerung		:= 0;
	fbPidLuftmengeVent1.Hold_I					:= FALSE;
	fbPidLuftmengeVent1.Hysterese				:= 0.0;
	fbPidLuftmengeVent1.Invert					:= FALSE;
	fbPidLuftmengeVent1.D_Anteil				:= Betriebsparameter.Ventilator1.D;
	fbPidLuftmengeVent1.D_Filterzeit			:= Betriebsparameter.Ventilator1.D * 1.4;
	fbPidLuftmengeVent1.I_Anteil				:= Betriebsparameter.Ventilator1.I;
	fbPidLuftmengeVent1.P_Anteil				:= Betriebsparameter.Ventilator1.P;
	fbPidLuftmengeVent1.RampeMax				:= 0.0;
	fbPidLuftmengeVent1.RegelbereichMin			:= Betriebsparameter.Sensoren.LuftgeschwMessberMin;
	IF Betriebsparameter.Ausstattung.Entfeuchter THEN
		fbPidLuftmengeVent1.RegelbereichMax		:= Betriebsparameter.Entfeuchter.LuftgeschwEntfeuchterMax;
	ELSE
		fbPidLuftmengeVent1.RegelbereichMax		:= Betriebsparameter.Sensoren.LuftgeschwMessberMax;
	END_IF
	fbPidLuftmengeVent1.StellgroesseManuell		:= 0.0;
	fbPidLuftmengeVent1.StellgroesseMin			:= Betriebsparameter.Ventilator1.DrehzahlMin;
	fbPidLuftmengeVent1.StellgroesseMax			:= Betriebsparameter.Ventilator1.DrehzahlMax;
	fbPidLuftmengeVent1.WindupDaempfung			:= 0.0;

	//====================================================================================================================================================================================
	//Luftmengenregler Ventilator 2 Eingänge
	//====================================================================================================================================================================================

	PidLuftmengeVent2.Sollgroesse				:= loc_LuftgeschwSollVent2;
	fbPidLuftmengeVent2.Freigabe				:= PidLuftmengeVent2.Enable;
	fbPidLuftmengeVent2.Sollwert				:= PidLuftmengeVent2.Sollgroesse;
	fbPidLuftmengeVent2.Istwert					:= gStatusAnlage.Luftgeschwindigkeit;
	fbPidLuftmengeVent2.AbschwaechungSollwert	:= 1.0;
	fbPidLuftmengeVent2.Aufschaltgroesse		:= 0.0;
	fbPidLuftmengeVent2.Fehlerverzoegerung		:= 0;
	fbPidLuftmengeVent2.Hold_I					:= FALSE;
	fbPidLuftmengeVent2.Hysterese				:= 0.0;
	fbPidLuftmengeVent2.Invert					:= FALSE;
	fbPidLuftmengeVent2.D_Anteil				:= Betriebsparameter.Ventilator2.D;
	fbPidLuftmengeVent2.D_Filterzeit			:= Betriebsparameter.Ventilator2.D * 1.4;
	fbPidLuftmengeVent2.I_Anteil				:= Betriebsparameter.Ventilator2.I;
	fbPidLuftmengeVent2.P_Anteil				:= Betriebsparameter.Ventilator2.P;
	fbPidLuftmengeVent2.RampeMax				:= 0.0;
	fbPidLuftmengeVent2.RegelbereichMin			:= Betriebsparameter.Sensoren.LuftgeschwMessberMin;
	IF Betriebsparameter.Ausstattung.Entfeuchter THEN
		fbPidLuftmengeVent1.RegelbereichMax		:= Betriebsparameter.Entfeuchter.LuftgeschwEntfeuchterMax;
	ELSE
		fbPidLuftmengeVent1.RegelbereichMax		:= Betriebsparameter.Sensoren.LuftgeschwMessberMax;
	END_IF
	fbPidLuftmengeVent2.StellgroesseManuell		:= 0.0;
	fbPidLuftmengeVent2.StellgroesseMin			:= Betriebsparameter.Ventilator2.DrehzahlMin;
	fbPidLuftmengeVent2.StellgroesseMax			:= Betriebsparameter.Ventilator2.DrehzahlMax;
	fbPidLuftmengeVent2.WindupDaempfung			:= 0.0;

	//====================================================================================================================================================================================
	//Drehzahlregelung Kompressor 1 Eingänge
	//====================================================================================================================================================================================

	PidKompressor1.Sollgroesse				:= Betriebsparameter.Kompressor1.NiederdruckSoll;
	fbPidKompressor1.Freigabe				:= PidKompressor1.Enable;
	fbPidKompressor1.Sollwert				:= PidKompressor1.Sollgroesse;
	fbPidKompressor1.Istwert				:= gStatusAnlage.NiederdruckModul1;
	fbPidKompressor1.AbschwaechungSollwert	:= 1.0;
	fbPidKompressor1.Aufschaltgroesse		:= 0.0;
	fbPidKompressor1.Fehlerverzoegerung		:= 0;
	fbPidKompressor1.Hold_I					:= FALSE;
	fbPidKompressor1.Hysterese				:= Betriebsparameter.Kompressor1.Hysterese;
	fbPidKompressor1.Invert					:= TRUE;
	fbPidKompressor1.D_Anteil				:= Betriebsparameter.Kompressor1.D;
	fbPidKompressor1.D_Filterzeit			:= Betriebsparameter.Kompressor1.D * 1.4;
	fbPidKompressor1.I_Anteil				:= Betriebsparameter.Kompressor1.I;
	fbPidKompressor1.P_Anteil				:= Betriebsparameter.Kompressor1.P;
	fbPidKompressor1.RampeMax				:= 0.0;
	fbPidKompressor1.RegelbereichMin		:= Betriebsparameter.Sensoren.NiederdruckMessberMin;
	fbPidKompressor1.RegelbereichMax		:= Betriebsparameter.Sensoren.NiederdruckMessberMax;
	fbPidKompressor1.StellgroesseManuell	:= 0.0;
	fbPidKompressor1.StellgroesseMin		:= Betriebsparameter.Kompressor1.DrehzahlMin;
	fbPidKompressor1.StellgroesseMax		:= Betriebsparameter.Kompressor1.DrehzahlMax;
	fbPidKompressor1.WindupDaempfung		:= 0.0;

	//====================================================================================================================================================================================
	//Drehzahlregelung Kompressor 2 Eingänge
	//====================================================================================================================================================================================

	PidKompressor2.Sollgroesse				:= Betriebsparameter.Kompressor2.NiederdruckSoll;
	fbPidKompressor2.Freigabe				:= PidKompressor2.Enable;
	fbPidKompressor2.Sollwert				:= PidKompressor2.Sollgroesse;
	fbPidKompressor2.Istwert				:= gStatusAnlage.NiederdruckModul2;
	fbPidKompressor2.AbschwaechungSollwert	:= 1.0;
	fbPidKompressor2.Aufschaltgroesse		:= 0.0;
	fbPidKompressor2.Fehlerverzoegerung		:= 0;
	fbPidKompressor2.Hold_I					:= FALSE;
	fbPidKompressor2.Hysterese				:= Betriebsparameter.Kompressor2.Hysterese;
	fbPidKompressor2.Invert					:= TRUE;
	fbPidKompressor2.D_Anteil				:= Betriebsparameter.Kompressor2.D;
	fbPidKompressor2.D_Filterzeit			:= Betriebsparameter.Kompressor2.D * 1.4;
	fbPidKompressor2.I_Anteil				:= Betriebsparameter.Kompressor2.I;
	fbPidKompressor2.P_Anteil				:= Betriebsparameter.Kompressor2.P;
	fbPidKompressor2.RampeMax				:= 0.0;
	fbPidKompressor2.RegelbereichMin		:= Betriebsparameter.Sensoren.NiederdruckMessberMin;
	fbPidKompressor2.RegelbereichMax		:= Betriebsparameter.Sensoren.NiederdruckMessberMax;
	fbPidKompressor2.StellgroesseManuell	:= 0.0;
	fbPidKompressor2.StellgroesseMin		:= Betriebsparameter.Kompressor2.DrehzahlMin;
	fbPidKompressor2.StellgroesseMax		:= Betriebsparameter.Kompressor2.DrehzahlMax;
	fbPidKompressor2.WindupDaempfung		:= 0.0;

	//====================================================================================================================================================================================
	//Heizregister-Regler Eingänge
	//====================================================================================================================================================================================

	PidHeizregister.Sollgroesse					:= Betriebsparameter.Heizregister.TrockenluftTempSoll;
	fbPidHeizregister.Freigabe					:= PidHeizregister.Enable;
	fbPidHeizregister.Sollwert					:= PidHeizregister.Sollgroesse;
	fbPidHeizregister.Istwert					:= gStatusAnlage.TrockenluftTemperatur;
	fbPidHeizregister.AbschwaechungSollwert		:= 1.0;
	fbPidHeizregister.Aufschaltgroesse			:= 0.0;
	fbPidHeizregister.Fehlerverzoegerung		:= 0;
	fbPidHeizregister.Hold_I					:= FALSE;
	fbPidHeizregister.Hysterese					:= Betriebsparameter.Heizregister.Hysterese;
	fbPidHeizregister.Invert					:= FALSE;
	fbPidHeizregister.D_Anteil					:= Betriebsparameter.Heizregister.D;
	fbPidHeizregister.D_Filterzeit				:= Betriebsparameter.Heizregister.D * 1.4;
	fbPidHeizregister.I_Anteil					:= Betriebsparameter.Heizregister.I;
	fbPidHeizregister.P_Anteil					:= Betriebsparameter.Heizregister.P;
	fbPidHeizregister.RampeMax					:= 0.0;
	fbPidHeizregister.RegelbereichMin			:= 0.0;
	fbPidHeizregister.RegelbereichMax			:= 100.0;
	fbPidHeizregister.StellgroesseManuell		:= 0.0;
	fbPidHeizregister.StellgroesseMin			:= Betriebsparameter.Heizregister.DrehzahlVorgabeMin;
	fbPidHeizregister.StellgroesseMax			:= Betriebsparameter.Heizregister.DrehzahlVorgabeMax;
	fbPidHeizregister.WindupDaempfung			:= 0.0;

	//====================================================================================================================================================================================
	//Abluftregler Eingänge
	//====================================================================================================================================================================================

	PidAbluftregler.Sollgroesse					:= Betriebsparameter.Abluftventilator.AbluftfeuchteMax;
	fbPidAbluftregler.Freigabe					:= PidAbluftregler.Enable;
	fbPidAbluftregler.Sollwert					:= PidAbluftregler.Sollgroesse;
	fbPidAbluftregler.Istwert					:= gStatusAnlage.AbluftFeuchte;
	fbPidAbluftregler.AbschwaechungSollwert		:= 1.0;
	fbPidAbluftregler.Aufschaltgroesse			:= 0.0;
	fbPidAbluftregler.Fehlerverzoegerung		:= 0;
	fbPidAbluftregler.Hold_I					:= FALSE;
	fbPidAbluftregler.Hysterese					:= Betriebsparameter.Abluftventilator.Hysterese;
	fbPidAbluftregler.Invert					:= TRUE;
	fbPidAbluftregler.D_Anteil					:= Betriebsparameter.Abluftventilator.D;
	fbPidAbluftregler.D_Filterzeit				:= Betriebsparameter.Abluftventilator.D * 1.4;
	fbPidAbluftregler.I_Anteil					:= Betriebsparameter.Abluftventilator.I;
	fbPidAbluftregler.P_Anteil					:= Betriebsparameter.Abluftventilator.P;
	fbPidAbluftregler.RampeMax					:= 0.0;
	fbPidAbluftregler.RegelbereichMin			:= 0.0;
	fbPidAbluftregler.RegelbereichMax			:= 100.0;
	fbPidAbluftregler.StellgroesseManuell		:= 0.0;
	fbPidAbluftregler.StellgroesseMin			:= Betriebsparameter.Abluftventilator.DrehzahlMin;
	fbPidAbluftregler.StellgroesseMax			:= Betriebsparameter.Abluftventilator.DrehzahlMax;
	fbPidAbluftregler.WindupDaempfung			:= 0.0;

	//========================================================================================================================================================================================
	//Schrittschaltwerk Regelung
	//========================================================================================================================================================================================

	//**********************************************************************************************************************************************************************************
	IF gAktModus = STILLSTAND THEN

		//*** Luftmengenregler Eingänge ***
		PidLuftmengeVent1.Enable	:= FALSE;
		PidLuftmengeVent2.Enable	:= FALSE;

		//*** Regler Kompressor 1 & 2 Eingänge ***
		PidKompressor1.Enable	:= FALSE;
		PidKompressor2.Enable	:= FALSE;

		//*** Regler Heizregister Eingänge ***
		PidHeizregister.Enable	:= FALSE;

		//*** Abluftregler Eingänge ***
		PidAbluftregler.Enable	:= Betriebsparameter.Abluftventilator.Automatik AND
		(Aktoren.VentUndKlappen.AnforderungVentilator1 OR Aktoren.VentUndKlappen.AnforderungVentilator2);

		//*** Drehzahlvorgabe Ventilator 1 & 2 ***
		IF Aktoren.VentUndKlappen.AnforderungVentilator1 THEN
			gCmdAnlage.Leistung.DrehzahlVentilator1	:= Betriebsparameter.Ventilator1.DrehzahlBeiAuskuehlphase;
		ELSE
			gCmdAnlage.Leistung.DrehzahlVentilator1	:= Betriebsparameter.Ventilator1.DrehzahlMin;
		END_IF

		IF Aktoren.VentUndKlappen.AnforderungVentilator2 THEN
			gCmdAnlage.Leistung.DrehzahlVentilator2	:= Betriebsparameter.Ventilator2.DrehzahlBeiAuskuehlphase;
		ELSE
			gCmdAnlage.Leistung.DrehzahlVentilator2	:= Betriebsparameter.Ventilator2.DrehzahlMin;
		END_IF

		//*** Drehzahlvorgabe Kompressor 1 & 2 ***
		gCmdAnlage.Leistung.DrehzahlKompressorModul1	:= 0.0;
		gCmdAnlage.Leistung.DrehzahlKompressorModul2	:= 0.0;

		//*** Drehzahlvorgabe Heizregister ***
		gCmdAnlage.Leistung.DrehzahlHeizregister		:= 0.0;

		//*** Drehzahlvorgabe Abluftventilator ***
		IF PidAbluftregler.Enable THEN
			gCmdAnlage.Leistung.DrehzahlAbluftventilator	:= fbPidAbluftregler.Stellgroesse;
		ELSE
			gCmdAnlage.Leistung.DrehzahlAbluftventilator	:= Betriebsparameter.Abluftventilator.DrehzahlMin;
		END_IF

		//**********************************************************************************************************************************************************************************
	ELSIF gAktModus = BETRIEB THEN

		//*** Luftmengenregler Eingänge ***
		//Kunde Gschneitner: Die Luftmengenregelung haengt an der Warmluft-/Kaltluftumschaltung des jeweiligen
		//Ventilators. Warmluft = Umluftlogik, dort kann der Bediener im Ventilator-Popup zwischen Fixdrehzahl
		//und Luftmengenregelung waehlen. Kaltluft = Frischluftlogik, dort ist in der Ausstattung nur die
		//Fixdrehzahl freigegeben, der Regler bleibt also aus.
		IF gStatusAnlage.Warmluft1 THEN
			PidLuftmengeVent1.Enable	:= Betriebsparameter.Ventilator1.LuftmengenregUmluftEin;
		ELSE
			PidLuftmengeVent1.Enable	:= Betriebsparameter.Ventilator1.LuftmengenregFrischluftEin;
		END_IF

		IF gStatusAnlage.Warmluft2 THEN
			PidLuftmengeVent2.Enable	:= Betriebsparameter.Ventilator2.LuftmengenregUmluftEin;
		ELSE
			PidLuftmengeVent2.Enable	:= Betriebsparameter.Ventilator2.LuftmengenregFrischluftEin;
		END_IF

		//Originallogik (Frischluft-/Umluftbetrieb) - fuer Kunde Gschneitner nicht in Verwendung:
		(*
		//*** Luftmengenregler Eingänge ***
		IF gStatusAnlage.FrischluftbetriebAktiv AND Betriebsparameter.Ventilator1.LuftmengenregFrischluftEin THEN
			PidLuftmengeVent1.Enable	:= TRUE;
		//ELSIF (gStatusAnlage.UmluftbetriebAktiv AND Betriebsparameter.Ventilator1.LuftmengenregUmluftEin) AND NOT hmiButtons.changeWarmluftVent1 THEN
		//	PidLuftmengeVent1.Enable	:= TRUE;
		//Kunde Gschneitner wenn Warmluftbetrieb Ventilator 1 aktiv dann Luftmengenregler aktivieren
		ELSIF hmiButtons.changeWarmluftVent1 THEN
			PidLuftmengeVent1.Enable	:= TRUE;
		ELSE
			PidLuftmengeVent1.Enable	:= FALSE;
		END_IF

		IF gStatusAnlage.FrischluftbetriebAktiv AND Betriebsparameter.Ventilator2.LuftmengenregFrischluftEin THEN
			PidLuftmengeVent2.Enable	:= TRUE;
		//ELSIF (gStatusAnlage.UmluftbetriebAktiv AND Betriebsparameter.Ventilator2.LuftmengenregUmluftEin) AND NOT hmiButtons.changeWarmluftVent2 THEN
		//	PidLuftmengeVent2.Enable	:= TRUE;
		//Kunde Gschneitner wenn Warmluftbetrieb Ventilator 2 aktiv dann Luftmengenregler aktivieren
		ELSIF hmiButtons.changeWarmluftVent2 THEN
			PidLuftmengeVent2.Enable	:= TRUE;
		ELSE
			PidLuftmengeVent2.Enable	:= FALSE;
		END_IF

		*)

		//*** Regler Kompressor 1 & 2 Eingänge ***
		PidKompressor1.Enable	:= Betriebsparameter.Kompressor1.DrehzahlregelungEin;
		PidKompressor2.Enable	:= Betriebsparameter.Kompressor2.DrehzahlregelungEin;

		//*** Regler Heizregister Eingänge ***
		//Kunde Gschneitner: Regler zusaetzlich sperren, wenn kein laufender Ventilator auf Warmluft steht
		//(sonst laeuft der I-Anteil weiter, waehrend das Heizregister bereits abgeschaltet ist).
		PidHeizregister.Enable	:= Betriebsparameter.Ausstattung.Heizregister AND NOT diHeizregisterFrostschutz AND
		gStatusAnlage.WarmluftAnforderung;

		//*** Abluftregler Eingänge ***
		PidAbluftregler.Enable	:= Betriebsparameter.Abluftventilator.Automatik;

		//*** Drehzahlvorgabe Ventilator 1 ***
		//Kunde Gschneitner: Fixdrehzahl je nach Stellung der Warmluft-/Kaltluftumschaltung des Ventilators.
		//Kaltluft = Frischluftlogik -> DrehzahlFixFrischluft, Warmluft = Umluftlogik -> DrehzahlFixUmluft.

		//Digitaler Eingang Leistungsreduzierung aktiv
		IF diDrehzahlbegrVentilator1 THEN
			IF PidLuftmengeVent1.Enable THEN
				IF (fbPidLuftmengeVent1.Stellgroesse > Betriebsparameter.Ventilator1.DrehzahlLeistungsreduz) THEN
					gCmdAnlage.Leistung.DrehzahlVentilator1	:= Betriebsparameter.Ventilator1.DrehzahlLeistungsreduz;
				ELSE
					gCmdAnlage.Leistung.DrehzahlVentilator1	:= fbPidLuftmengeVent1.Stellgroesse;
				END_IF
			ELSIF (NOT gStatusAnlage.Warmluft1) THEN
				IF (Betriebsparameter.Ventilator1.DrehzahlFixFrischluft > Betriebsparameter.Ventilator1.DrehzahlLeistungsreduz) THEN
					gCmdAnlage.Leistung.DrehzahlVentilator1	:= Betriebsparameter.Ventilator1.DrehzahlLeistungsreduz;
				ELSE
					gCmdAnlage.Leistung.DrehzahlVentilator1	:= Betriebsparameter.Ventilator1.DrehzahlFixFrischluft;
				END_IF
			ELSIF gStatusAnlage.Warmluft1 THEN
				IF (Betriebsparameter.Ventilator1.DrehzahlFixUmluft > Betriebsparameter.Ventilator1.DrehzahlLeistungsreduz) THEN
					gCmdAnlage.Leistung.DrehzahlVentilator1	:= Betriebsparameter.Ventilator1.DrehzahlLeistungsreduz;
				ELSE
					gCmdAnlage.Leistung.DrehzahlVentilator1	:= Betriebsparameter.Ventilator1.DrehzahlFixUmluft;
				END_IF
			END_IF
			//Strombegrenzung aktiv (Zeitfenster)
		ELSIF Strombegrenzung.StrombegrenzungEin THEN
			IF PidLuftmengeVent1.Enable THEN
				IF (fbPidLuftmengeVent1.Stellgroesse > Betriebsparameter.Ventilator1.DrehzahlStrombegrenzung) THEN
					gCmdAnlage.Leistung.DrehzahlVentilator1	:= Betriebsparameter.Ventilator1.DrehzahlStrombegrenzung;
				ELSE
					gCmdAnlage.Leistung.DrehzahlVentilator1	:= fbPidLuftmengeVent1.Stellgroesse;
				END_IF
			ELSIF (NOT gStatusAnlage.Warmluft1) THEN
				IF (Betriebsparameter.Ventilator1.DrehzahlFixFrischluft > Betriebsparameter.Ventilator1.DrehzahlStrombegrenzung) THEN
					gCmdAnlage.Leistung.DrehzahlVentilator1	:= Betriebsparameter.Ventilator1.DrehzahlStrombegrenzung;
				ELSE
					gCmdAnlage.Leistung.DrehzahlVentilator1	:= Betriebsparameter.Ventilator1.DrehzahlFixFrischluft;
				END_IF
			ELSIF gStatusAnlage.Warmluft1 THEN
				IF (Betriebsparameter.Ventilator1.DrehzahlFixUmluft > Betriebsparameter.Ventilator1.DrehzahlStrombegrenzung) THEN
					gCmdAnlage.Leistung.DrehzahlVentilator1	:= Betriebsparameter.Ventilator1.DrehzahlStrombegrenzung;
				ELSE
					gCmdAnlage.Leistung.DrehzahlVentilator1	:= Betriebsparameter.Ventilator1.DrehzahlFixUmluft;
				END_IF
			END_IF
		//Notbetrieb Ventilator -> Drehzahl Auskühlphase
		ELSIF (Boxen.NotbetriebVentilator1 AND NOT Boxen.FreigabeVentilator1) THEN
			gCmdAnlage.Leistung.DrehzahlVentilator1 := Betriebsparameter.Ventilator1.DrehzahlBeiAuskuehlphase;
			//Luftmengenregelung aktiv
		ELSIF PidLuftmengeVent1.Enable THEN
			gCmdAnlage.Leistung.DrehzahlVentilator1	:= fbPidLuftmengeVent1.Stellgroesse;
			//Betrieb mit Fixdrehzahlen
		ELSE
			IF (NOT gStatusAnlage.Warmluft1) THEN
				gCmdAnlage.Leistung.DrehzahlVentilator1	:= Betriebsparameter.Ventilator1.DrehzahlFixFrischluft;
			ELSE
				gCmdAnlage.Leistung.DrehzahlVentilator1	:= Betriebsparameter.Ventilator1.DrehzahlFixUmluft;
			END_IF
		END_IF

		//*** Drehzahlvorgabe Ventilator 2 ***
		//Kunde Gschneitner: Fixdrehzahl je nach Stellung der Warmluft-/Kaltluftumschaltung des Ventilators.
		//Kaltluft = Frischluftlogik -> DrehzahlFixFrischluft, Warmluft = Umluftlogik -> DrehzahlFixUmluft.

		//Digitaler Eingang Leistungsreduzierung aktiv
		IF diDrehzahlbegrVentilator2 THEN
			IF PidLuftmengeVent2.Enable THEN
				IF (fbPidLuftmengeVent2.Stellgroesse > Betriebsparameter.Ventilator2.DrehzahlLeistungsreduz) THEN
					gCmdAnlage.Leistung.DrehzahlVentilator2	:= Betriebsparameter.Ventilator2.DrehzahlLeistungsreduz;
				ELSE
					gCmdAnlage.Leistung.DrehzahlVentilator2	:= fbPidLuftmengeVent2.Stellgroesse;
				END_IF
			ELSIF (NOT gStatusAnlage.Warmluft2) THEN
				IF (Betriebsparameter.Ventilator2.DrehzahlFixFrischluft > Betriebsparameter.Ventilator2.DrehzahlLeistungsreduz) THEN
					gCmdAnlage.Leistung.DrehzahlVentilator2	:= Betriebsparameter.Ventilator2.DrehzahlLeistungsreduz;
				ELSE
					gCmdAnlage.Leistung.DrehzahlVentilator2	:= Betriebsparameter.Ventilator2.DrehzahlFixFrischluft;
				END_IF
			ELSIF gStatusAnlage.Warmluft2 THEN
				IF (Betriebsparameter.Ventilator2.DrehzahlFixUmluft > Betriebsparameter.Ventilator2.DrehzahlLeistungsreduz) THEN
					gCmdAnlage.Leistung.DrehzahlVentilator2	:= Betriebsparameter.Ventilator2.DrehzahlLeistungsreduz;
				ELSE
					gCmdAnlage.Leistung.DrehzahlVentilator2	:= Betriebsparameter.Ventilator2.DrehzahlFixUmluft;
				END_IF
			END_IF
			//Strombegrenzung aktiv (Zeitfenster)
		ELSIF Strombegrenzung.StrombegrenzungEin THEN
			IF PidLuftmengeVent2.Enable THEN
				IF (fbPidLuftmengeVent2.Stellgroesse > Betriebsparameter.Ventilator2.DrehzahlStrombegrenzung) THEN
					gCmdAnlage.Leistung.DrehzahlVentilator2	:= Betriebsparameter.Ventilator2.DrehzahlStrombegrenzung;
				ELSE
					gCmdAnlage.Leistung.DrehzahlVentilator2	:= fbPidLuftmengeVent2.Stellgroesse;
				END_IF
			ELSIF (NOT gStatusAnlage.Warmluft2) THEN
				IF (Betriebsparameter.Ventilator2.DrehzahlFixFrischluft > Betriebsparameter.Ventilator2.DrehzahlStrombegrenzung) THEN
					gCmdAnlage.Leistung.DrehzahlVentilator2	:= Betriebsparameter.Ventilator2.DrehzahlStrombegrenzung;
				ELSE
					gCmdAnlage.Leistung.DrehzahlVentilator2	:= Betriebsparameter.Ventilator2.DrehzahlFixFrischluft;
				END_IF
			ELSIF gStatusAnlage.Warmluft2 THEN
				IF (Betriebsparameter.Ventilator2.DrehzahlFixUmluft > Betriebsparameter.Ventilator2.DrehzahlStrombegrenzung) THEN
					gCmdAnlage.Leistung.DrehzahlVentilator2	:= Betriebsparameter.Ventilator2.DrehzahlStrombegrenzung;
				ELSE
					gCmdAnlage.Leistung.DrehzahlVentilator2	:= Betriebsparameter.Ventilator2.DrehzahlFixUmluft;
				END_IF
			END_IF
		//Notbetrieb Ventilator -> Drehzahl Auskühlphase
		ELSIF (Boxen.NotbetriebVentilator2 AND NOT Boxen.FreigabeVentilator2) THEN
			gCmdAnlage.Leistung.DrehzahlVentilator2 := Betriebsparameter.Ventilator2.DrehzahlBeiAuskuehlphase;
			//Luftmengenregelung aktiv
		ELSIF PidLuftmengeVent2.Enable THEN
			gCmdAnlage.Leistung.DrehzahlVentilator2	:= fbPidLuftmengeVent2.Stellgroesse;
			//Betrieb mit Fixdrehzahlen
		ELSE
			IF (NOT gStatusAnlage.Warmluft2) THEN
				gCmdAnlage.Leistung.DrehzahlVentilator2	:= Betriebsparameter.Ventilator2.DrehzahlFixFrischluft;
			ELSE
				gCmdAnlage.Leistung.DrehzahlVentilator2	:= Betriebsparameter.Ventilator2.DrehzahlFixUmluft;
			END_IF
		END_IF

		//*** Drehzahlvorgabe Kompressor 1 ***

		//Digitaler Eingang für Leistungsreduzierung aktiv
		IF diLeistungsvorgKompressorExtMod1 THEN
			IF PidKompressor1.Enable THEN
				IF fbPidKompressor1.Stellgroesse > Betriebsparameter.Kompressor1.DrehzahlReduzierung THEN
					gCmdAnlage.Leistung.DrehzahlKompressorModul1	:= Betriebsparameter.Kompressor1.DrehzahlReduzierung;
				ELSE
					gCmdAnlage.Leistung.DrehzahlKompressorModul1	:= fbPidKompressor1.Stellgroesse;
				END_IF
			END_IF
		//Drehzahlregelung aktiv
		ELSIF PidKompressor1.Enable THEN
			gCmdAnlage.Leistung.DrehzahlKompressorModul1	:= fbPidKompressor1.Stellgroesse;
		//Betrieb mit Fixdrehzahl
		ELSE
			gCmdAnlage.Leistung.DrehzahlKompressorModul1	:= Betriebsparameter.Kompressor1.DrehzahlFix;
		END_IF

		//*** Drehzahlvorgabe Kompressor 2 ***

		//Digitaler Eingang für Leistungsreduzierung aktiv
		IF diLeistungsvorgKompressorExtMod1 THEN
			IF PidKompressor2.Enable THEN
				IF fbPidKompressor2.Stellgroesse > Betriebsparameter.Kompressor2.DrehzahlReduzierung THEN
					gCmdAnlage.Leistung.DrehzahlKompressorModul2	:= Betriebsparameter.Kompressor2.DrehzahlReduzierung;
				ELSE
					gCmdAnlage.Leistung.DrehzahlKompressorModul2	:= fbPidKompressor2.Stellgroesse;
				END_IF
			END_IF
			//Drehzahlregelung aktiv
		ELSIF PidKompressor2.Enable THEN
			gCmdAnlage.Leistung.DrehzahlKompressorModul2	:= fbPidKompressor2.Stellgroesse;
			//Betrieb mit Fixdrehzahl
		ELSE
			gCmdAnlage.Leistung.DrehzahlKompressorModul2	:= Betriebsparameter.Kompressor2.DrehzahlFix;
		END_IF

		//*** Drehzahlvorgabe Heizregister ***
		IF PidHeizregister.Enable AND Aktoren.Heizregister.FreigabeHeizregisterOut THEN
			gCmdAnlage.Leistung.DrehzahlHeizregister		:= fbPidHeizregister.Stellgroesse;
		ELSE
			gCmdAnlage.Leistung.DrehzahlHeizregister		:= Betriebsparameter.Heizregister.DrehzahlVorgabeMin;
		END_IF

		//*** Drehzahlvorgabe Abluftventilator ***
		IF gStatusAnlage.FrischluftbetriebAktiv AND Betriebsparameter.Ausstattung.AbluftklImFrischlbetrImmerOffen THEN
			gCmdAnlage.Leistung.DrehzahlAbluftventilator	:= Betriebsparameter.Abluftventilator.DrehzahlMax;
		ELSIF PidAbluftregler.Enable AND Betriebsparameter.Abluftventilator.Automatik THEN
			gCmdAnlage.Leistung.DrehzahlAbluftventilator	:= fbPidAbluftregler.Stellgroesse;
		ELSE
			gCmdAnlage.Leistung.DrehzahlAbluftventilator	:= Betriebsparameter.Abluftventilator.DrehzahlMax;
		END_IF

	//***************************************************************************************************************************************************************
	ELSE

		//*** Luftmengenregler Eingänge ***
		PidLuftmengeVent1.Enable	:= FALSE;
		PidLuftmengeVent2.Enable	:= FALSE;

		//*** Regler Kompressor 1 & 2 Eingänge ***
		PidKompressor1.Enable	:= FALSE;
		PidKompressor2.Enable	:= FALSE;

		//*** Regler Heizregister Eingänge ***
		PidHeizregister.Enable	:= FALSE;

		//*** Abluftregler Eingänge ***
		PidAbluftregler.Enable	:= FALSE;

		//*** Drehzahlvorgabe Ventilator 1 & 2 ***
		gCmdAnlage.Leistung.DrehzahlVentilator1	:= 0.0;
		gCmdAnlage.Leistung.DrehzahlVentilator2	:= 0.0;

		//*** Drehzahlvorgabe Kompressor 1 & 2 ***
		gCmdAnlage.Leistung.DrehzahlKompressorModul1	:= 0.0;
		gCmdAnlage.Leistung.DrehzahlKompressorModul2	:= 0.0;

		//*** Drehzahlvorgabe Heizregister ***
		gCmdAnlage.Leistung.DrehzahlHeizregister		:= 0.0;

		//*** Drehzahlvorgabe Abluftventilator ***
		gCmdAnlage.Leistung.DrehzahlAbluftventilator	:= 0.0;

	END_IF

	//Funktionsblock Aufrufe
	//=======================

	//Luftmengenregler Ventilator 1
	IF fbPidLuftmengeVent1.Freigabe THEN
		fbPidLuftmengeVent1.Mode	:= FBREG_MODUS_AUTO;
	ELSE
		fbPidLuftmengeVent1.Mode	:= FBREG_MODUS_FREEZE;
	END_IF
	fbPidLuftmengeVent1();

	//Luftmengenregler Ventilator 2
	IF fbPidLuftmengeVent2.Freigabe THEN
		fbPidLuftmengeVent2.Mode	:= FBREG_MODUS_AUTO;
	ELSE
		fbPidLuftmengeVent2.Mode	:= FBREG_MODUS_FREEZE;
	END_IF
	fbPidLuftmengeVent2();

	//Regler Heizregister
	IF fbPidHeizregister.Freigabe THEN
		fbPidHeizregister.Mode	:= FBREG_MODUS_AUTO;
	ELSE
		fbPidHeizregister.Mode	:= FBREG_MODUS_FREEZE;
	END_IF
	fbPidHeizregister();

	//Regler Kompressor 1
	IF fbPidKompressor1.Freigabe THEN
		fbPidKompressor1.Mode	:= FBREG_MODUS_AUTO;
	ELSE
		fbPidKompressor1.Mode	:= FBREG_MODUS_FREEZE;
	END_IF
	fbPidKompressor1();

	//Regler Kompressor 2
	IF fbPidKompressor2.Freigabe THEN
		fbPidKompressor2.Mode	:= FBREG_MODUS_AUTO;
	ELSE
		fbPidKompressor2.Mode	:= FBREG_MODUS_FREEZE;
	END_IF
	fbPidKompressor2();

	//Abluftregler
	IF fbPidAbluftregler.Freigabe THEN
		fbPidAbluftregler.Mode	:= FBREG_MODUS_AUTO;
	ELSE
		fbPidAbluftregler.Mode	:= FBREG_MODUS_FREEZE;
	END_IF
	fbPidAbluftregler();

END_PROGRAM
```

#### Leistung.var - Lokale Variablen
```iecst
VAR
	fbLascoZdxx_0 : {REDUND_UNREPLICABLE} fbLascoZdxx;
	fbLascoZdxx_1 : {REDUND_UNREPLICABLE} fbLascoZdxx;
	sekTick : {REDUND_UNREPLICABLE} BOOL;
	minTick : {REDUND_UNREPLICABLE} BOOL;
	loc_LuftgeschwSollVent1 : {REDUND_UNREPLICABLE} REAL;
	loc_LuftgeschwSollVent2 : {REDUND_UNREPLICABLE} REAL;
	fbBoxenLuftmengen_0 : {REDUND_UNREPLICABLE} fbBoxenLuftmengen;
	loc_Ansaugflaeche : {REDUND_UNREPLICABLE} REAL;
	loc_LuftmengeSollKaltVent1 : {REDUND_UNREPLICABLE} REAL; (*Kunde Gschneitner: Soll-Luftmenge Ventilator 1 mit den Frischluft-Parametern (Kaltluft)*)
	loc_LuftmengeSollKaltVent2 : {REDUND_UNREPLICABLE} REAL; (*Kunde Gschneitner: Soll-Luftmenge Ventilator 2 mit den Frischluft-Parametern (Kaltluft)*)
	loc_LuftmengeSollWarmVent1 : {REDUND_UNREPLICABLE} REAL; (*Kunde Gschneitner: Soll-Luftmenge Ventilator 1 mit den Umluft-Parametern (Warmluft)*)
	loc_LuftmengeSollWarmVent2 : {REDUND_UNREPLICABLE} REAL; (*Kunde Gschneitner: Soll-Luftmenge Ventilator 2 mit den Umluft-Parametern (Warmluft)*)
END_VAR
```

### RegelungIO.var - Paket Variablen
```iecst
VAR
	PidLuftmengeVent1 : typ_PidControl;
	PidLuftmengeVent2 : typ_PidControl;
	PidKompressor1 : typ_PidControl;
	PidKompressor2 : typ_PidControl;
	PidHeizregister : typ_PidControl;
	PidAbluftregler : typ_PidControl;
	fbPidLuftmengeVent1 : fbRegPidReglerAllg;
	fbPidLuftmengeVent2 : fbRegPidReglerAllg;
	fbPidKompressor1 : fbRegPidReglerAllg;
	fbPidKompressor2 : fbRegPidReglerAllg;
	fbPidHeizregister : fbRegPidReglerAllg;
	fbPidAbluftregler : fbRegPidReglerAllg;
END_VAR
```

### RegelungIO.typ - Paket Datentypen
```iecst
TYPE
	typ_PidControl : 	STRUCT
		Enable : BOOL;
		Sollgroesse : REAL;
		Stellgroesse : REAL;
		FehlerReglerMax : BOOL;
		FehlerReglerMin : BOOL;
		WarnungReglerMax : BOOL;
		WarnungReglerMin : BOOL;
	END_STRUCT;
END_TYPE
```

- Visualisation Logical/Visualisierung (not shown)

### Package Logical/CSV - Paket Datenaufzeichnung

### CSV_Global.typ
```iecst
TYPE
	CSV_typ : 	STRUCT
		IW : CSV_IW_typ;
		SW : CSV_SW_typ;
		FE : CSV_FE_typ;
		WA : CSV_WA_typ;
	END_STRUCT;
	CSV_IW_typ : 	STRUCT
		RPS_SAVE_STEP_Nr : UINT;
		RPS_CPYDEL_STEP_Nr : UINT;
		RPS_SAVE_STEP_Text : STRING[80];
		RPS_CPYDEL_STEP_Text : STRING[80];
		SFehler : BOOL;
		SFehler_Nr : USINT;
		SWarnung : BOOL;
		SWarnung_Nr : USINT;
		KOPF_WRITE : BOOL;
		DATA_WRITE : BOOL;
		DATA_WRITE_BEREIT : BOOL;
		Zyklus_t_akt : UDINT;
		Zyklus_t_letzt : UDINT;
		DatObj_Zeilen_Anz : UINT;
		DatObj_Tag_ID_ZeileNr : UINT;
		DatObj_Tag_Variable_ZeileNr : UINT;
		DatObj_Tag_Datentyp_ZeileNr : UINT;
		DatObj_Tag_MIN_ZeileNr : UINT;
		DatObj_Tag_MAX_ZeileNr : UINT;
		RPS_DirRead_Start_OK : BOOL;
		RPS_COPY_AUTO_Start : BOOL;
		DirRead_FileName_alt : STRING[260];
		DirRead_FileName_neu : STRING[260];
		PC_DevLink_Param : STRING[200];
		PC_Device : STRING[20];
		PC_Zielpfad : STRING[100];
		EXT_Device : STRING[20];
		EXT_Zielpfad : STRING[100];
		RPS_Device : ARRAY[0..19] OF USINT;
		RPS_Zielpfad : ARRAY[0..19] OF USINT;
		RPS_DirCreate_OK : BOOL;
		RPS_FileCreate_OK : BOOL;
		RPS_FileOpen_OK : BOOL;
		RPS_FileWrite_OK : BOOL;
		RPS_FileRead_OK : BOOL;
		RPS_FileClose_OK : BOOL;
		RPS_MemInfo_OK : BOOL;
		RPS_DirInfo_OK : BOOL;
		RPS_DirRead_OK : BOOL;
		RPS_FileDelete_OK : BOOL;
		RPS_DirDeleteEx_OK : BOOL;
		PC_DevLink_OK : BOOL;
		PC_DirCreate_OK : BOOL;
		PC_FileCopy_OK : BOOL;
		PC_DirCopy_OK : BOOL;
		EXT_DirCreate_OK : BOOL;
		EXT_FileCopy_OK : BOOL;
		EXT_DirCopy_OK : BOOL;
		RPS_DirCreate_FehlerNr : UINT;
		RPS_FileCreate_FehlerNr : UINT;
		RPS_FileOpen_FehlerNr : UINT;
		RPS_FileWrite_FehlerNr : UINT;
		RPS_FileRead_FehlerNr : UINT;
		RPS_FileClose_FehlerNr : UINT;
		RPS_MemInfo_FehlerNr : UINT;
		RPS_DirInfo_FehlerNr : UINT;
		RPS_DirRead_FehlerNr : UINT;
		RPS_FileDelete_FehlerNr : UINT;
		RPS_DirCopy_FehlerNr : UINT;
		RPS_DirDeleteEx_FehlerNr : UINT;
		PC_DevLink_FehlerNr : UINT;
		PC_DirCreate_FehlerNr : UINT;
		PC_FileCopy_FehlerNr : UINT;
		PC_DirCopy_FehlerNr : UINT;
		EXT_DirCreate_FehlerNr : UINT;
		EXT_FileCopy_FehlerNr : UINT;
		EXT_DirCopy_FehlerNr : UINT;
		RPS_DirCreate_OK_Z : UDINT;
		RPS_DirCreate_FEHLER_Z : UDINT;
		RPS_FileCreate_OK_Z : UDINT;
		RPS_FileCreate_FEHLER_Z : UDINT;
		RPS_FileOpen_OK_Z : UDINT;
		RPS_FileOpen_FEHLER_Z : UDINT;
		RPS_FileWrite_OK_Z : UDINT;
		RPS_FileWrite_FEHLER_Z : UDINT;
		RPS_FileRead_OK_Z : UDINT;
		RPS_FileRead_FEHLER_Z : UDINT;
		RPS_FileClose_OK_Z : UDINT;
		RPS_FileClose_FEHLER_Z : UDINT;
		RPS_MemInfo_OK_Z : UDINT;
		RPS_MemInfo_FEHLER_Z : UDINT;
		RPS_DirInfo_OK_Z : UDINT;
		RPS_DirInfo_FEHLER_Z : UDINT;
		RPS_DirRead_OK_Z : UDINT;
		RPS_DirRead_FEHLER_Z : UDINT;
		RPS_FileDelete_OK_Z : UDINT;
		RPS_FileDelete_FEHLER_Z : UDINT;
		RPS_DirDeleteEx_OK_Z : UDINT;
		RPS_DirDeleteEx_FEHLER_Z : UDINT;
		PC_DevLink_OK_Z : UDINT;
		PC_DevLink_FEHLER_Z : UDINT;
		PC_DirCreate_OK_Z : UDINT;
		PC_DirCreate_FEHLER_Z : UDINT;
		PC_FileCopy_OK_Z : UDINT;
		PC_FileCopy_FEHLER_Z : UDINT;
		PC_DirCopy_OK_Z : UDINT;
		PC_DirCopy_FEHLER_Z : UDINT;
		EXT_DirCreate_OK_Z : UDINT;
		EXT_DirCreate_FEHLER_Z : UDINT;
		EXT_FileCopy_OK_Z : UDINT;
		EXT_FileCopy_FEHLER_Z : UDINT;
		EXT_DirCopy_OK_Z : UDINT;
		EXT_DirCopy_FEHLER_Z : UDINT;
		Version : ARRAY[0..19] OF USINT;
		Anlagename : ARRAY[0..19] OF USINT;
		File_Name : STRING[100];
		RPS_File_Name : STRING[200];
		RPS_Mem_frei : UDINT;
		RPS_Mem_frei_prz : REAL;
		RPS_Mem_gesamt : UDINT;
		RPS_DirInfo_FileNum : UDINT;
		RPS_DirInfo_DirNum : UDINT;
		RPS_DirRead_Data : fiDIR_READ_DATA;
		Kopf_length : UDINT;
		Datensatz_length : UDINT;
		Datensatz_TimeStamp : ARRAY[0..24] OF USINT;
	END_STRUCT;
	CSV_SW_typ : 	STRUCT
		SPERRE_T : BOOL;
		KOPF_WRITE_T : BOOL;
		DATA_WRITE_T : BOOL;
		F_Quitt_T : BOOL;
		Gruebl_Reporting_T : BOOL;
		QM_HeizW_T : BOOL;
		QM_HeizW_BetrJahr_Mon : USINT;
		Kopf_Version_T : BOOL;
		Kopf_Anlagenname_T : BOOL;
		Kopf_ID_T : BOOL;
		Kopf_Bezeichnung_T : BOOL;
		Kopf_Einheit_T : BOOL;
		Kopf_Datentyp_T : BOOL;
		Kopf_MIN_MAX_T : BOOL;
		Zeitstempel_lang_T : BOOL;
		Begrenzung_MINMAX_T : BOOL;
		RPS_Mem_frei_przN : REAL;
		RPS_COPY_AUTO_T : BOOL;
		RPS_MEMORY_AUTO_T : BOOL;
		RPS_FileDelete_alt_HAND_T : BOOL;
		RPS_FileDelete_neu_HAND_T : BOOL;
		RPS_DirDeleteEx_HAND_T : BOOL;
		PC_FileCopy_alt_HAND_T : BOOL;
		PC_FileCopy_neu_HAND_T : BOOL;
		PC_DirCopy_HAND_T : BOOL;
		EXT_FileCopy_alt_HAND_T : BOOL;
		EXT_FileCopy_neu_HAND_T : BOOL;
		EXT_DirCopy_HAND_T : BOOL;
	END_STRUCT;
	CSV_FE_typ : 	STRUCT
		Datensatz_Fehler : BOOL;
		DatObj_CFG : BOOL;
		DatObj_CFG_length : BOOL;
		DatObj_Tag_ID : BOOL;
		DatObj_Tag_Variable : BOOL;
		DatObj_Tag_Datentyp : BOOL;
		DatObj_Tag_MIN : BOOL;
		DatObj_Tag_MAX : BOOL;
		DatObj_ZeilenMAX : BOOL;
		RPS_kein_Speicherplatz : BOOL;
		RPS_DirCreate : BOOL;
		RPS_FileCreate : BOOL;
		RPS_FileOpen : BOOL;
		RPS_FileClose : BOOL;
		RPS_FileWrite : BOOL;
		RPS_FileRead : BOOL;
		RPS_MemInfo : BOOL;
		RPS_DirInfo : BOOL;
		RPS_DirRead : BOOL;
		RPS_FileDelete : BOOL;
		RPS_DirDeleteEx : BOOL;
		PC_DevLink : BOOL;
		PC_DirCreate : BOOL;
		PC_FileCopy : BOOL;
		PC_DirCopy : BOOL;
		EXT_DirCreate : BOOL;
		EXT_FileCopy : BOOL;
		EXT_DirCopy : BOOL;
	END_STRUCT;
	CSV_WA_typ : 	STRUCT
		RPS_Datei_alt_geloescht : BOOL;
		File_not_found : BOOL;
	END_STRUCT;
	CSV_DatObj1_typ : 	STRUCT
		Version : ARRAY[0..19] OF USINT;
		Anlagename : ARRAY[0..19] OF USINT;
		RPS_Device : ARRAY[0..19] OF USINT;
		RPS_Zielpfad : ARRAY[0..19] OF USINT;
		EXT_Device : ARRAY[0..19] OF USINT;
		EXT_Zielpfad : ARRAY[0..19] OF USINT;
		PC_IP_Adresse : ARRAY[0..19] OF USINT;
		PC_Ordnerfreigabe : ARRAY[0..19] OF USINT;
		PC_Username : ARRAY[0..19] OF USINT;
		PC_Userpassword : ARRAY[0..19] OF USINT;
		PC_Zielpfad : ARRAY[0..99] OF USINT;
	END_STRUCT;
	CSV_DatObj2_typ : 	STRUCT
		Tag_ID : DINT;
		Tag_Variablenname : ARRAY[0..47] OF USINT;
		Tag_Bezeichnung : ARRAY[0..59] OF USINT;
		Tag_Einheit : ARRAY[0..31] OF USINT;
		Tag_MIN : ARRAY[0..15] OF USINT;
		Tag_MAX : ARRAY[0..15] OF USINT;
	END_STRUCT;
END_TYPE
```

### CSV_Global.var
```iecst
VAR
	device_param : STRING[80] := '';
	device_name : STRING[80];
END_VAR
VAR RETAIN
	CSV01 : CSV_typ;
	CSV_Uhr : DTStructure;
	CSV_Uhr_Sp : DTStructure;
END_VAR
```

### Library Logical/CSV/Library/CSV (IEC, version 1.00.0) - CSV Library

#### CSV.fun - Exported functions and function blocks
```iecst
(********************************************************************
 * COPYRIGHT --
 ********************************************************************
 * Library: CSV01
 * File: CSV01.fun
 * Author: Herwig
 * Created: February 24, 2011
 ********************************************************************
 * Functions and function blocks of library CSV01
 ********************************************************************)

FUNCTION_BLOCK CSV_Tick
	VAR_INPUT
		Enable : BOOL;
		Wert : REAL;
	END_VAR
	VAR_OUTPUT
		Ausg : BOOL;
	END_VAR
	VAR
		SpWert : REAL;
	END_VAR
END_FUNCTION_BLOCK

FUNCTION_BLOCK CSV_itoa
	VAR_INPUT
		Eing_DINT : DINT;
		Eing_Anz_VK : USINT;
		Eing_Anz_NK : USINT;
		Eing_Vorz_Plus : BOOL;
		Eing_Komma_Punkt : BOOL;
		Ausg_ASCII_adr : UDINT;
		Ausg_ASCII_len : UDINT;
	END_VAR
	VAR_OUTPUT
		Ausg_Fehler : BOOL;
	END_VAR
	VAR
		Eing_DINT_VK : DINT;
		Eing_DINT_NK : DINT;
		Str_VK_len : UINT;
		Str_NK_len : UINT;
		Str_Ges_len : UINT;
		Str_VK : ARRAY[0..11] OF USINT;
		Str_NK : ARRAY[0..11] OF USINT;
		M_ASCII : ARRAY[0..24] OF USINT;
		i : USINT;
	END_VAR
END_FUNCTION_BLOCK

FUNCTION_BLOCK CSV_GRP_date
	VAR_INPUT
		Eing_Tag : USINT;
		Eing_Monat : USINT;
		Eing_Jahr : UINT;
		Ausg_date_adr : UDINT;
		Ausg_date_len : UDINT;
	END_VAR
	VAR_OUTPUT
		Ausg_Fehler : BOOL;
	END_VAR
	VAR
		M_DATE : ARRAY[0..10] OF USINT;
		Str_Jahr : ARRAY[0..11] OF USINT;
		Str_Mon : ARRAY[0..11] OF USINT;
		Str_Tag : ARRAY[0..11] OF USINT;
		M_Fehler : BOOL;
		zzCSV_itoa00000 : CSV_itoa;
		zzCSV_itoa00001 : CSV_itoa;
		zzCSV_itoa00002 : CSV_itoa;
	END_VAR
END_FUNCTION_BLOCK

FUNCTION_BLOCK CSV_GRP_time
	VAR_INPUT
		Eing_Stunde : USINT;
		Eing_Minute : USINT;
		Eing_Sekunde : USINT;
		Ausg_time_adr : UDINT;
		Ausg_time_len : UDINT;
	END_VAR
	VAR_OUTPUT
		Ausg_Fehler : BOOL;
	END_VAR
	VAR
		M_TIME : ARRAY[0..8] OF USINT;
		Str_Stunde : ARRAY[0..11] OF USINT;
		Str_Minute : ARRAY[0..11] OF USINT;
		Str_Sekunde : ARRAY[0..11] OF USINT;
		M_Fehler : BOOL;
		zzCSV_itoa00000 : CSV_itoa;
		zzCSV_itoa00001 : CSV_itoa;
		zzCSV_itoa00002 : CSV_itoa;
	END_VAR
END_FUNCTION_BLOCK

FUNCTION_BLOCK CSV_GRP_timestamp
	VAR_INPUT
		Eing_Tag : USINT;
		Eing_Monat : USINT;
		Eing_Jahr : UINT;
		Eing_Stunde : USINT;
		Eing_Minute : USINT;
		Eing_Sekunde : USINT;
		Eing_MilliSek : UINT;
		Ausg_timestamp_adr : UDINT;
		Ausg_timestamp_len : UDINT;
	END_VAR
	VAR_OUTPUT
		Ausg_Fehler : BOOL;
	END_VAR
	VAR
		M_TIMESTAMP : ARRAY[0..23] OF USINT;
		Str_Jahr : ARRAY[0..11] OF USINT;
		Str_Mon : ARRAY[0..11] OF USINT;
		Str_Tag : ARRAY[0..11] OF USINT;
		Str_Stunde : ARRAY[0..11] OF USINT;
		Str_Minute : ARRAY[0..11] OF USINT;
		Str_Sekunde : ARRAY[0..11] OF USINT;
		Str_MilliSek : ARRAY[0..11] OF USINT;
		M_Fehler : BOOL;
		zzCSV_itoa00000 : CSV_itoa;
		zzCSV_itoa00001 : CSV_itoa;
		zzCSV_itoa00002 : CSV_itoa;
		zzCSV_itoa00003 : CSV_itoa;
		zzCSV_itoa00004 : CSV_itoa;
		zzCSV_itoa00005 : CSV_itoa;
		zzCSV_itoa00006 : CSV_itoa;
	END_VAR
END_FUNCTION_BLOCK

FUNCTION_BLOCK CSV_QM_timestamp
	VAR_INPUT
		Eing_Tag : USINT;
		Eing_Monat : USINT;
		Eing_Jahr : UINT;
		Eing_Stunde : USINT;
		Eing_Minute : USINT;
		Ausg_timestamp_adr : UDINT;
		Ausg_timestamp_len : UDINT;
	END_VAR
	VAR_OUTPUT
		Ausg_Fehler : BOOL;
	END_VAR
	VAR
		M_TIMESTAMP : ARRAY[0..14] OF USINT;
		Str_Tag : ARRAY[0..11] OF USINT;
		Str_Mon : ARRAY[0..11] OF USINT;
		Str_Jahr : ARRAY[0..11] OF USINT;
		Str_Stunde : ARRAY[0..11] OF USINT;
		Str_Minute : ARRAY[0..11] OF USINT;
		M_Fehler : BOOL;
		zzCSV_itoa00000 : CSV_itoa;
		zzCSV_itoa00001 : CSV_itoa;
		zzCSV_itoa00002 : CSV_itoa;
		zzCSV_itoa00003 : CSV_itoa;
		zzCSV_itoa00004 : CSV_itoa;
	END_VAR
END_FUNCTION_BLOCK

FUNCTION_BLOCK CSV_atoLREAL
	VAR_INPUT
		Eing_ASCII_adr : UDINT;
		Eing_ASCII_len : UDINT;
	END_VAR
	VAR_OUTPUT
		Ausg_Fehler : BOOL;
		Ausg_LREAL : LREAL;
	END_VAR
	VAR
		M_ASCII : ARRAY[0..40] OF USINT;
		ii : USINT;
		M_Stellen : SINT;
		M_Vorkomma : SINT;
		M_Komma : BOOL;
	END_VAR
END_FUNCTION_BLOCK

FUNCTION_BLOCK CSV_UDINTtoa
	VAR_INPUT
		Eing_UDINT : UDINT;
		Ausg_ASCII_adr : UDINT;
		Ausg_ASCII_len : UDINT;
	END_VAR
	VAR_OUTPUT
		Ausg_Fehler : BOOL;
	END_VAR
	VAR
		Ausg_ASCII : ARRAY[0..10] OF USINT;
		i : SINT;
		ii : SINT;
		M_Start : BOOL;
	END_VAR
END_FUNCTION_BLOCK
```

#### CSV_Tick.ab
```automation-basic
FUNCTION_BLOCK CSV_Tick
;====================================================================
;                   FUB: CSV_Tick
;
;	Aufruf:	CSV_Tick ( Enable, Wert,   Ausg  )
;				       Bool    Real   Bool
;
; 	Author:		Ing. Schmid Herwig
;	Version:	1.0
;	Datum:	    24.02.2011
;	geprüft:	24.02.2011 OK
;====================================================================
;
; Fkt:	Gibt bei Enable = 1 und einer Wertänderung von "Wert" EINEN Impuls "Ausg" aus
;====================================================================

  if Enable = 0 then
	SpWert = Wert
	Ausg = 0
  else If (Wert <> SpWert) then
	Ausg = 1
	SpWert = Wert
  else
	Ausg = 0
  endif

END_FUNCTION_BLOCK
```

#### CSV_itoa.ab
```automation-basic
;====================================================================
;                  DINT-Wert wird in ASCII gewandelt
;     Vorzeichenoption, Vor-Nachkommastellen, Kommazeichen können
;     definiert werden. Damit können genau formatierte Strings erzeugt werden
;       z.B.: Eing_DINT =     1, Eing_Anz_NK = 3, Eing_Anz_VK = 4, Eing_Vorz_Plus = 0, Eing_Komma_Punkt = 1  :  Ausg = "0000.001"
;       z.B.: Eing_DINT =   123, Eing_Anz_NK = 1, Eing_Anz_VK = 0, Eing_Vorz_Plus = 0, Eing_Komma_Punkt = 1  :  Ausg = "12.3"
;       z.B.: Eing_DINT = -1234, Eing_Anz_NK = 2, Eing_Anz_VK = 5, Eing_Vorz_Plus = 1, Eing_Komma_Punkt = 0  :  Ausg = "-00012,34"
;       z.B.: Eing_DINT =    -4, Eing_Anz_NK = 2, Eing_Anz_VK = 3, Eing_Vorz_Plus = 1, Eing_Komma_Punkt = 0  :  Ausg = "+000,04"
;       z.B.: Eing_DINT =  1234, Eing_Anz_NK = 2, Eing_Anz_VK = 1, Eing_Vorz_Plus = 1, Eing_Komma_Punkt = 0  :  Ausg = "+2,34"
;
;   !!  Achtung: Angeschlossener String muß mindestens die Zeichen der angegebenen Stellen incl. Vorzeichen + Komma haben ansonsten wird ein Fehler ausgegeben
;                String[12] bzw. USINT[0..12] notwendig für DINT z.B.: -214748364.8
;
; 	Author:		Ing. Schmid Herwig
;	Version:	1.0
;	Datum:		08.03.2011
;	geprüft:	08.03.2011 OK
;
;====================================================================
; Aufruf: CSV_itoa(Eing_DINT, Eing_Anz_VK, Eing_Anz_NK, Eing_Vorz_Plus, Eing_Komma_Punkt, adr(Ausg_ASCII), sizeof(Ausg_ASCII), Ausg_Fehler)
;
; EA:    		Eing_DINT 		  	  E.. DINT Eingangswert -2147483648..+2147483647
;               Eing_Anz_NK           E.. USINT <=9  Anzahl der Nachkomma-Stellen (sind am Eingang weniger Stellen vorhanden als Nachkomma definiert, so wird nach dem Komma mit "0" aufgefüllt)
;               Eing_Anz_VK           E.. USINT <=10 Anzahl der Vorkomma-Stellen  (bleiben weniger Vorkomma über als hier angegeben, so wird vorne mit "0" aufgefüllt)
;               Eing_Vorz_Plus        E.. BOOL (1= bei positiven Zahlen wird "+" vorangestellt)
;               Eing_Komma_Punkt      E.. BOOL Definition des Kommazeichens (0=, 1=.)
;              	adr(Ausg_ASCII)	  	  E.. Adresse von USINT[>=0..10] od. STRING[>=10]
;              	sizeof(Ausg_ASCII) 	  E.. Länge von USINT[>=0..10] od. STRING[>=10]
;              	Ausg_Fehler           A.. BOOL (= 1 wenn String od. USINT zu klein definiert)
;====================================================================

FUNCTION_BLOCK CSV_itoa

; Vor- und Nachkommazahl trennen und in String wandeln:
  Eing_DINT_VK = Eing_DINT / DINT(EXPT(10, Eing_Anz_NK))
  Eing_DINT_NK = Eing_DINT - Eing_DINT_VK * DINT(EXPT(10, Eing_Anz_NK))
  memset(adr(Str_VK) , 0, sizeof(Str_VK))
  memset(adr(Str_NK) , 0, sizeof(Str_NK))
  memset(adr(M_ASCII), 0, sizeof(M_ASCII))
  Str_VK_len = itoa(ABS(Eing_DINT_VK), adr(Str_VK)) ; Vorzeichen weglassen
  Str_NK_len = itoa(ABS(Eing_DINT_NK), adr(Str_NK)) ; Vorzeichen weglassen

  if Eing_Anz_VK >= Str_VK_len then
     Str_Ges_len = UINT(Eing_Anz_VK + Eing_Anz_NK)
  else
     Str_Ges_len = UINT(Str_VK_len + Eing_Anz_NK)
  endif
  if (Eing_Anz_NK > 0) then
     Str_Ges_len = Str_Ges_len + 1	; zusätzliche Stelle für Komma
  endif
  if (Eing_Vorz_Plus = 1) or (Eing_DINT < 0) then
     Str_Ges_len = Str_Ges_len + 1	; zusätzliche Stelle für Vorzeichen
  endif

  if (Str_Ges_len <= Ausg_ASCII_len) and (Eing_Anz_VK <= 10) and (Eing_Anz_NK <= 9) then   ; max 12 Stellen erlaubt bzw. möglich: z.B.: -214748364.7

	Ausg_Fehler = 0

; Nachkomma-String: Bei Bedarf restliche Stellen vorne mit "0" auffüllen:
     if Str_NK_len < Eing_Anz_NK then
        loop i = Eing_Anz_NK-1 downto 0 do
             if i >= Eing_Anz_NK-Str_NK_len then
		        Str_NK[i] = Str_NK[i-(Eing_Anz_NK-Str_NK_len)]
	         else
		        Str_NK[i] = 48
		     endif
        endloop
     endif

; Vorkomma-String: Bei Bedarf restliche Stellen vorne mit "0" auffüllen:
     if Str_VK_len < Eing_Anz_VK then
        loop i = Eing_Anz_VK-1 downto 0 do
             if i >= Eing_Anz_VK-Str_VK_len then
		        Str_VK[i] = Str_VK[i-(Eing_Anz_VK-Str_VK_len)]
	         else
		        Str_VK[i] = 48
		     endif
        endloop
     endif

; Vorzeichen je nach Modus hizufügen:
     if (Eing_DINT < 0) then
        M_ASCII[0] = 45  ;"-"
     else if (Eing_Vorz_Plus = 1)  then
        M_ASCII[0] = 43  ;"+"
     endif

; ASCII-String zusammenfügen und bei Bedarf Komma "," od. "." setzen:
     strcat(adr(M_ASCII), adr(Str_VK))
     if Eing_Anz_NK > 0 then
        if Eing_Komma_Punkt = 1 then
	       strcat(adr(M_ASCII), ".")
	    else
	       strcat(adr(M_ASCII), ",")
        endif
        strcat(adr(M_ASCII), adr(Str_NK))
     endif

  else

  	Ausg_Fehler = 1

  endif

  if Ausg_ASCII_len >= sizeof(M_ASCII) then
     memcpy(Ausg_ASCII_adr, adr(M_ASCII), sizeof(M_ASCII))
  else
     memcpy(Ausg_ASCII_adr, adr(M_ASCII), Ausg_ASCII_len)
  endif

END_FUNCTION_BLOCK
```

#### CSV_GRP_date.ab - Date-Konvertierung für Grübl-Reporting Software
```automation-basic
;====================================================================
;        Eingangswerte Tag, Monat, Jahr in einen formatierten String für
;              Grübl-Reporting (GRP) Format: "jjjj-MM-dd" umwandeln
;
;   !!  Achtung: mindestens String[10] od. USINT[0..10] am Ausgang anhängen !!
;
;       (Auffüllung Tage < 10, Monat < 10, Jahr < 1000 mit vorangestellten "0")
;        zB.: "2011-01-01"
;
; 	Author:		Ing. Schmid Herwig
;	Version:	1.0
;	Datum:		25.02.2011
;	geprüft:	25.02.2011 OK
;
;====================================================================
; Aufruf: CSV_GRP_date(Eing_Tag, Eing_Monat, Eing_Jahr, adr(Ausg_date), sizeof(Ausg_date), Ausg_Fehler)
;
; EA:    		Eing_Tag  		  E.. Byte     Tageswert 1..31
;              	Eing_Monat	  	  E.. Byte     Monatswert 1..12
;              	Eing_Jahr         E.. UINT     Jahreswert 0..9999
;              	adr(Ausg_date)	  E.. UDINT    Ausgangsvariable - Adresse String[>=10] od. USINT[>=0..10]
;               sizeof(Ausg_date) E.. UDINT    Ausgangsvariable - Länge String[>=10] od. USINT[>=0..10]
;               Ausg_Fehler       A.. BOOL     (= 1 wenn Ausgangsvariable zu klein definiert)
;====================================================================

FUNCTION_BLOCK CSV_GRP_date

  memset(adr(M_DATE), 0, sizeof(M_DATE))

  if Ausg_date_len >= sizeof(M_DATE) then

     CSV_itoa(Eing_Tag  , 2, 0, 0, 0, adr(Str_Tag) , sizeof(Str_Tag) , M_Fehler)
     CSV_itoa(Eing_Monat, 2, 0, 0, 0, adr(Str_Mon) , sizeof(Str_Mon) , M_Fehler)
     CSV_itoa(Eing_Jahr , 4, 0, 0, 0, adr(Str_Jahr), sizeof(Str_Jahr), M_Fehler)

     strcpy(adr(M_DATE), adr(Str_Jahr))
     strcat(adr(M_DATE), "-")
     strcat(adr(M_DATE), adr(Str_Mon))
     strcat(adr(M_DATE), "-")
     strcat(adr(M_DATE), adr(Str_Tag))

     memcpy(Ausg_date_adr, adr(M_DATE), Ausg_date_len)

  else

    memcpy(Ausg_date_adr, adr(M_DATE), sizeof(M_DATE))
  	Ausg_Fehler = 1

  endif

END_FUNCTION_BLOCK
```

#### CSV_GRP_time.ab - Time-Konvertierung für Grübl-Reporting Software
```automation-basic
;====================================================================
;              Eingangswerte Stunde, Minute, Sekunde in einen String für
;              Grübl-Reporting (GRP) Format: "hh:mm:ss" umwandeln
;
;   !!  Achtung: mindestens String[8] od. USINT[0..8] am Ausgang anhängen !!
;
;       (Auffüllung Stunde < 10, Minute < 10, Sekunde < 10 mit vorangestellten "0")
;        zB.: "05:35:09"
;
; 	Author:		Ing. Schmid Herwig
;	Version:	1.0
;	Datum:		25.02.2011
;	geprüft:	25.02.2011 OK
;
;====================================================================
; Aufruf: CSV_GRP_time(Eing_Stunde, Eing_Minute, Eing_Sekunde, adr(Ausg_time), sizeof(Ausg_time), Ausg_Fehler)
;
; EA:    		Eing_Stunde  	  E.. Byte    Stundenwert  0..23
;              	Eing_Minute	  	  E.. Byte    Minutenwert  0..59
;              	Eing_Sekunde      E.. UINT    Sekundenwert 0..59
;              	adr(Ausg_time)	  E.. UDINT   Ausgangsvariable - Adresse String[>=8] od. USINT[>=0..8]
;               sizeof(Ausg_time) E.. UDINT   Ausgangsvariable - Länge String[>=8] od. USINT[>=0..8]
;               Ausg_Fehler       A.. BOOL    (= 1 wenn Ausgangsvariable zu klein definiert)
;====================================================================

FUNCTION_BLOCK CSV_GRP_time

  memset(adr(M_TIME), 0, sizeof(M_TIME))

  if Ausg_time_len >= sizeof(M_TIME) then

     CSV_itoa(Eing_Stunde , 2, 0, 0, 0, adr(Str_Stunde) , sizeof(Str_Stunde),  M_Fehler)
     CSV_itoa(Eing_Minute , 2, 0, 0, 0, adr(Str_Minute) , sizeof(Str_Minute),  M_Fehler)
     CSV_itoa(Eing_Sekunde, 2, 0, 0, 0, adr(Str_Sekunde), sizeof(Str_Sekunde), M_Fehler)

     strcpy(adr(M_TIME), adr(Str_Stunde))
     strcat(adr(M_TIME), ":")
     strcat(adr(M_TIME), adr(Str_Minute))
     strcat(adr(M_TIME), ":")
     strcat(adr(M_TIME), adr(Str_Sekunde))

     memcpy(Ausg_time_adr, adr(M_TIME), Ausg_time_len)

  else

    memcpy(Ausg_time_adr, adr(M_TIME), sizeof(M_TIME))
  	Ausg_Fehler = 1

  endif

END_FUNCTION_BLOCK
```

#### CSV_GRP_timestamp.ab - Timestamp-Konvertierung für Grübl-Reporting Software
```automation-basic
;====================================================================
; Eingangswerte Tag, Monat, Jahr, Stunde, Minute, Sekunde, MilliSek in einen String für
; Grübl-Reporting (GRP) Format: "jjjj-MM-dd hh:mm:ss.nnn" umwandeln
;
;   !!  Achtung: mindestens String[23] od. USINT[0..23] am Ausgang anhängen !!
;
;       (Auffüllung Tage < 10, Monat < 10, Jahr < 1000
;                   Stunde < 10, Minute < 10, Sekunde < 10 milliSek < 10 mit vorangestellten "0")
;        zB.: "2011-01-01 09:35:27.365"
;
; 	Author:		Ing. Schmid Herwig
;	Version:	1.0
;	Datum:		25.02.2011
;	geprüft:	25.02.2011 OK
;
;====================================================================
; Aufruf: CSV_GRP_timestamp(Eing_Tag, Eing_Monat, Eing_Jahr, Eing_Stunde, Eing_Minute, Eing_Sekunde, Eing_MilliSek, adr(Ausg_timestamp), sizeof(Ausg_timestamp), Ausg_Fehler)
;
; EA:    		Eing_Tag  		  	   E.. Byte   Tageswert    1..31
;              	Eing_Monat	  	  	   E.. Byte   Monatswert   1..12
;              	Eing_Jahr        	   E.. UINT   Jahreswert   0..9999
;               Eing_Stunde  	  	   E.. Byte   Stundenwert  0..23
;              	Eing_Minute	  	  	   E.. Byte   Minutenwert  0..59
;              	Eing_Sekunde      	   E.. UINT   Sekundenwert 0..59
;              	Eing_MilliSek     	   E.. UINT   Sekundenwert 0..999
;              	adr(Ausg_timestamp)	   E.. UDINT  Ausgangsvariable - Adresse String[>=23] od. USINT[>=0..23]
;               sizeof(Ausg_timestamp) E.. UDINT  Ausgangsvariable - Länge String[>=23] od. USINT[>=0..23]
;               Ausg_Fehler            A.. BOOL   (= 1 wenn Ausgangsvariable zu klein definiert)
;====================================================================

FUNCTION_BLOCK CSV_GRP_timestamp

  memset(adr(M_TIMESTAMP), 0, sizeof(M_TIMESTAMP))

  if Ausg_timestamp_len >= sizeof(M_TIMESTAMP) then

     CSV_itoa(Eing_Tag  , 2, 0, 0, 0, adr(Str_Tag) , sizeof(Str_Tag) , M_Fehler)
     CSV_itoa(Eing_Monat, 2, 0, 0, 0, adr(Str_Mon) , sizeof(Str_Mon) , M_Fehler)
     CSV_itoa(Eing_Jahr , 4, 0, 0, 0, adr(Str_Jahr), sizeof(Str_Jahr), M_Fehler)

     CSV_itoa(Eing_Stunde  , 2, 0, 0, 0, adr(Str_Stunde)  , sizeof(Str_Stunde),   M_Fehler)
     CSV_itoa(Eing_Minute  , 2, 0, 0, 0, adr(Str_Minute)  , sizeof(Str_Minute),   M_Fehler)
     CSV_itoa(Eing_Sekunde , 2, 0, 0, 0, adr(Str_Sekunde) , sizeof(Str_Sekunde),  M_Fehler)
     CSV_itoa(Eing_MilliSek, 3, 0, 0, 0, adr(Str_MilliSek), sizeof(Str_MilliSek), M_Fehler)

     strcpy(adr(M_TIMESTAMP), adr(Str_Jahr))
     strcat(adr(M_TIMESTAMP), "-")
     strcat(adr(M_TIMESTAMP), adr(Str_Mon))
     strcat(adr(M_TIMESTAMP), "-")
     strcat(adr(M_TIMESTAMP), adr(Str_Tag))
     strcat(adr(M_TIMESTAMP), " ")
     strcat(adr(M_TIMESTAMP), adr(Str_Stunde))
     strcat(adr(M_TIMESTAMP), ":")
     strcat(adr(M_TIMESTAMP), adr(Str_Minute))
     strcat(adr(M_TIMESTAMP), ":")
     strcat(adr(M_TIMESTAMP), adr(Str_Sekunde))
     strcat(adr(M_TIMESTAMP), ".")
     strcat(adr(M_TIMESTAMP), adr(Str_MilliSek))

     memcpy(Ausg_timestamp_adr, adr(M_TIMESTAMP), Ausg_timestamp_len)

  else

     memcpy(Ausg_timestamp_adr, adr(M_TIMESTAMP), sizeof(M_TIMESTAMP))
  	 Ausg_Fehler = 1

  endif

END_FUNCTION_BLOCK
```
